LIN {X 0.013,Y -527.446,Z 1176.432,A 0.000,B 0.000,C 90.000,E1 293.695} C_DIS
LIN {X -0.104,Y -527.276,Z 1176.422,A 0.000,B 0.000,C 90.000,E1 291.972} C_DIS
LIN {X -0.041,Y -526.939,Z 1176.411,A 0.000,B 0.000,C 90.000,E1 289.939} C_DIS
LIN {X 0.315,Y -526.514,Z 1176.400,A 0.000,B 0.000,C 90.000,E1 287.873} C_DIS
LIN {X 0.154,Y -526.111,Z 1176.393,A 0.000,B 0.000,C 90.000,E1 286.732} C_DIS
LIN {X -0.007,Y -525.425,Z 1176.385,A 0.000,B 0.000,C 90.000,E1 285.300} C_DIS
LIN {X 0.178,Y -524.796,Z 1176.379,A 0.000,B 0.000,C 90.000,E1 284.120} C_DIS
LIN {X -0.133,Y -523.544,Z 1176.369,A 0.000,B 0.000,C 90.000,E1 282.411} C_DIS
LIN {X -0.073,Y -522.465,Z 1176.359,A 0.000,B 0.000,C 90.000,E1 280.658} C_DIS
LIN {X -0.130,Y -521.579,Z 1176.351,A 0.000,B 0.000,C 90.000,E1 279.208} C_DIS
LIN {X -0.200,Y -520.907,Z 1176.345,A 0.000,B 0.000,C 90.000,E1 278.049} C_DIS
LIN {X 0.164,Y -520.008,Z 1176.337,A 0.000,B 0.000,C 90.000,E1 276.549} C_DIS
LIN {X -0.094,Y -518.805,Z 1176.325,A 0.000,B 0.000,C 90.000,E1 274.531} C_DIS
LIN {X 0.047,Y -517.732,Z 1176.314,A 0.000,B 0.000,C 90.000,E1 272.465} C_DIS
LIN {X 0.205,Y -516.891,Z 1176.304,A 0.000,B 0.000,C 90.000,E1 270.688} C_DIS
LIN {X -0.117,Y -516.202,Z 1176.296,A 0.000,B 0.000,C 90.000,E1 269.255} C_DIS
LIN {X 0.077,Y -515.566,Z 1176.288,A 0.000,B 0.000,C 90.000,E1 267.764} C_DIS
LIN {X -0.182,Y -514.943,Z 1176.281,A 0.000,B 0.000,C 90.000,E1 266.617} C_DIS
LIN {X 0.060,Y -514.072,Z 1176.275,A 0.000,B 0.000,C 90.000,E1 265.412} C_DIS
LIN {X 0.158,Y -512.347,Z 1176.263,A 0.000,B 0.000,C 90.000,E1 263.337} C_DIS
LIN {X -0.115,Y -511.308,Z 1176.257,A 0.000,B 0.000,C 90.000,E1 262.186} C_DIS
LIN {X 0.088,Y -509.594,Z 1176.247,A 0.000,B 0.000,C 90.000,E1 260.387} C_DIS
LIN {X 0.256,Y -507.511,Z 1176.234,A 0.000,B 0.000,C 90.000,E1 257.993} C_DIS
LIN {X 0.024,Y -505.767,Z 1176.222,A 0.000,B 0.000,C 90.000,E1 255.936} C_DIS
LIN {X -0.079,Y -504.700,Z 1176.215,A 0.000,B 0.000,C 90.000,E1 254.755} C_DIS
LIN {X -0.135,Y -503.462,Z 1176.207,A 0.000,B 0.000,C 90.000,E1 253.268} C_DIS
LIN {X 0.005,Y -501.999,Z 1176.197,A 0.000,B 0.000,C 90.000,E1 251.456} C_DIS
LIN {X 0.107,Y -500.375,Z 1176.187,A 0.000,B 0.000,C 90.000,E1 249.645} C_DIS
LIN {X -0.012,Y -498.966,Z 1176.179,A 0.000,B 0.000,C 90.000,E1 248.156} C_DIS
LIN {X -0.149,Y -497.507,Z 1176.170,A 0.000,B 0.000,C 90.000,E1 246.666} C_DIS
LIN {X -0.113,Y -495.810,Z 1176.162,A 0.000,B 0.000,C 90.000,E1 245.153} C_DIS
LIN {X -0.154,Y -494.396,Z 1176.155,A 0.000,B 0.000,C 90.000,E1 243.948} C_DIS
LIN {X 0.036,Y -492.401,Z 1176.147,A 0.000,B 0.000,C 90.000,E1 242.410} C_DIS
LIN {X 0.249,Y -489.559,Z 1176.135,A 0.000,B 0.000,C 90.000,E1 240.255} C_DIS
LIN {X 0.138,Y -487.469,Z 1176.126,A 0.000,B 0.000,C 90.000,E1 238.742} C_DIS
LIN {X 0.051,Y -484.871,Z 1176.116,A 0.000,B 0.000,C 90.000,E1 236.914} C_DIS
LIN {X 0.000,Y -480.986,Z 1176.101,A 0.000,B 0.000,C 90.000,E1 234.149} C_DIS
LIN {X 0.010,Y -478.812,Z 1176.092,A 0.000,B 0.000,C 90.000,E1 232.603} C_DIS
LIN {X -0.040,Y -475.824,Z 1176.080,A 0.000,B 0.000,C 90.000,E1 230.436} C_DIS
LIN {X 0.186,Y -473.842,Z 1176.072,A 0.000,B 0.000,C 90.000,E1 228.852} C_DIS
LIN {X 0.153,Y -472.537,Z 1176.066,A 0.000,B 0.000,C 90.000,E1 227.919} C_DIS
LIN {X -0.220,Y -467.466,Z 1176.047,A 0.000,B 0.000,C 90.000,E1 224.514} C_DIS
LIN {X 0.002,Y -464.713,Z 1176.033,A 0.000,B 0.000,C 90.000,E1 221.962} C_DIS
LIN {X -0.242,Y -462.501,Z 1176.007,A 0.000,B 0.000,C 90.000,E1 217.237} C_DIS
LIN {X 0.183,Y -462.031,Z 1175.991,A 0.000,B 0.000,C 90.000,E1 214.326} C_DIS
LIN {X 0.188,Y -462.258,Z 1175.980,A 0.000,B 0.000,C 90.000,E1 212.418} C_DIS
LIN {X 0.101,Y -463.482,Z 1175.968,A 0.000,B 0.000,C 90.000,E1 210.207} C_DIS
LIN {X 0.219,Y -465.265,Z 1175.956,A 0.000,B 0.000,C 90.000,E1 207.975} C_DIS
LIN {X -0.022,Y -468.504,Z 1175.938,A 0.000,B 0.000,C 90.000,E1 204.847} C_DIS
LIN {X 0.229,Y -475.785,Z 1175.914,A 0.000,B 0.000,C 90.000,E1 200.429} C_DIS
LIN {X 0.047,Y -484.654,Z 1175.893,A 0.000,B 0.000,C 90.000,E1 196.732} C_DIS
LIN {X 0.270,Y -493.798,Z 1175.876,A 0.000,B 0.000,C 90.000,E1 193.647} C_DIS
LIN {X 0.236,Y -500.640,Z 1175.864,A 0.000,B 0.000,C 90.000,E1 191.535} C_DIS
LIN {X -0.107,Y -505.714,Z 1175.856,A 0.000,B 0.000,C 90.000,E1 190.074} C_DIS
LIN {X -0.136,Y -514.040,Z 1175.843,A 0.000,B 0.000,C 90.000,E1 187.701} C_DIS
LIN {X 0.119,Y -519.246,Z 1175.835,A 0.000,B 0.000,C 90.000,E1 186.201} C_DIS
LIN {X -0.147,Y -526.357,Z 1175.823,A 0.000,B 0.000,C 90.000,E1 184.188} C_DIS
LIN {X -0.258,Y -532.477,Z 1175.814,A 0.000,B 0.000,C 90.000,E1 182.465} C_DIS
LIN {X -0.257,Y -539.492,Z 1175.802,A 0.000,B 0.000,C 90.000,E1 180.458} C_DIS
LIN {X -0.180,Y -543.585,Z 1175.796,A 0.000,B 0.000,C 90.000,E1 179.312} C_DIS
LIN {X 0.012,Y -548.578,Z 1175.788,A 0.000,B 0.000,C 90.000,E1 177.879} C_DIS
LIN {X 0.242,Y -552.555,Z 1175.782,A 0.000,B 0.000,C 90.000,E1 176.731} C_DIS
LIN {X 0.160,Y -558.479,Z 1175.773,A 0.000,B 0.000,C 90.000,E1 175.065} C_DIS
LIN {X 0.251,Y -564.346,Z 1175.764,A 0.000,B 0.000,C 90.000,E1 173.394} C_DIS
LIN {X -0.105,Y -570.116,Z 1175.754,A 0.000,B 0.000,C 90.000,E1 171.781} C_DIS
LIN {X 0.183,Y -574.902,Z 1175.747,A 0.000,B 0.000,C 90.000,E1 170.387} C_DIS
LIN {X -0.226,Y -578.690,Z 1175.741,A 0.000,B 0.000,C 90.000,E1 169.342} C_DIS
LIN {X -0.011,Y -584.216,Z 1175.732,A 0.000,B 0.000,C 90.000,E1 167.701} C_DIS
LIN {X 0.069,Y -588.852,Z 1175.724,A 0.000,B 0.000,C 90.000,E1 166.353} C_DIS
LIN {X -0.205,Y -593.226,Z 1175.717,A 0.000,B 0.000,C 90.000,E1 165.046} C_DIS
LIN {X 0.170,Y -597.631,Z 1175.709,A 0.000,B 0.000,C 90.000,E1 163.685} C_DIS
LIN {X -0.073,Y -601.090,Z 1175.704,A 0.000,B 0.000,C 90.000,E1 162.653} C_DIS
LIN {X 0.127,Y -604.447,Z 1175.698,A 0.000,B 0.000,C 90.000,E1 161.583} C_DIS
LIN {X -0.087,Y -608.460,Z 1175.691,A 0.000,B 0.000,C 90.000,E1 160.296} C_DIS
LIN {X 0.351,Y -612.366,Z 1175.683,A 0.000,B 0.000,C 90.000,E1 158.954} C_DIS
LIN {X -0.260,Y -615.395,Z 1175.678,A 0.000,B 0.000,C 90.000,E1 157.975} C_DIS
LIN {X -0.330,Y -620.612,Z 1175.667,A 0.000,B 0.000,C 90.000,E1 156.177} C_DIS
LIN {X 0.220,Y -624.160,Z 1175.660,A 0.000,B 0.000,C 90.000,E1 154.845} C_DIS
LIN {X 0.033,Y -628.945,Z 1175.651,A 0.000,B 0.000,C 90.000,E1 153.076} C_DIS
LIN {X -0.134,Y -631.608,Z 1175.645,A 0.000,B 0.000,C 90.000,E1 152.076} C_DIS
LIN {X 0.040,Y -634.839,Z 1175.638,A 0.000,B 0.000,C 90.000,E1 150.795} C_DIS
LIN {X 0.059,Y -638.466,Z 1175.629,A 0.000,B 0.000,C 90.000,E1 149.282} C_DIS
LIN {X -0.072,Y -641.780,Z 1175.621,A 0.000,B 0.000,C 90.000,E1 147.788} C_DIS
LIN {X -0.056,Y -643.800,Z 1175.615,A 0.000,B 0.000,C 90.000,E1 146.786} C_DIS
LIN {X -0.201,Y -645.736,Z 1175.610,A 0.000,B 0.000,C 90.000,E1 145.801} C_DIS
LIN {X 0.169,Y -648.438,Z 1175.602,A 0.000,B 0.000,C 90.000,E1 144.276} C_DIS
LIN {X 0.007,Y -650.641,Z 1175.595,A 0.000,B 0.000,C 90.000,E1 143.050} C_DIS
LIN {X -0.048,Y -652.350,Z 1175.589,A 0.000,B 0.000,C 90.000,E1 142.065} C_DIS
LIN {X 0.257,Y -654.569,Z 1175.582,A 0.000,B 0.000,C 90.000,E1 140.803} C_DIS
LIN {X 0.097,Y -657.952,Z 1175.573,A 0.000,B 0.000,C 90.000,E1 139.094} C_DIS
LIN {X -0.028,Y -661.068,Z 1175.565,A 0.000,B 0.000,C 90.000,E1 137.634} C_DIS
LIN {X 0.357,Y -664.130,Z 1175.557,A 0.000,B 0.000,C 90.000,E1 136.134} C_DIS
LIN {X 0.346,Y -669.386,Z 1175.543,A 0.000,B 0.000,C 90.000,E1 133.704} C_DIS
LIN {X -0.468,Y -673.988,Z 1175.532,A 0.000,B 0.000,C 90.000,E1 131.838} C_DIS
LIN {X -0.097,Y -679.759,Z 1175.519,A 0.000,B 0.000,C 90.000,E1 129.402} C_DIS
LIN {X -0.135,Y -683.328,Z 1175.511,A 0.000,B 0.000,C 90.000,E1 127.971} C_DIS
LIN {X -0.262,Y -686.330,Z 1175.504,A 0.000,B 0.000,C 90.000,E1 126.790} C_DIS
LIN {X 0.389,Y -689.886,Z 1175.496,A 0.000,B 0.000,C 90.000,E1 125.311} C_DIS
LIN {X -0.098,Y -692.169,Z 1175.491,A 0.000,B 0.000,C 90.000,E1 124.405} C_DIS
LIN {X 0.018,Y -694.299,Z 1175.486,A 0.000,B 0.000,C 90.000,E1 123.452} C_DIS
LIN {X -0.180,Y -696.901,Z 1175.479,A 0.000,B 0.000,C 90.000,E1 122.291} C_DIS
LIN {X 0.000,Y -698.834,Z 1175.474,A 0.000,B 0.000,C 90.000,E1 121.337} C_DIS
LIN {X 0.194,Y -700.659,Z 1175.469,A 0.000,B 0.000,C 90.000,E1 120.384} C_DIS
LIN {X 0.389,Y -701.877,Z 1175.465,A 0.000,B 0.000,C 90.000,E1 119.667} C_DIS
LIN {X -0.074,Y -703.846,Z 1175.459,A 0.000,B 0.000,C 90.000,E1 118.537} C_DIS
LIN {X 0.110,Y -705.271,Z 1175.453,A 0.000,B 0.000,C 90.000,E1 117.590} C_DIS
LIN {X 0.355,Y -706.061,Z 1175.449,A 0.000,B 0.000,C 90.000,E1 116.873} C_DIS
LIN {X -0.051,Y -706.576,Z 1175.444,A 0.000,B 0.000,C 90.000,E1 115.976} C_DIS
LIN {X -0.111,Y -706.732,Z 1175.440,A 0.000,B 0.000,C 90.000,E1 115.283} C_DIS
LIN {X -0.163,Y -706.601,Z 1175.438,A 0.000,B 0.000,C 90.000,E1 114.823} C_DIS
LIN {X -0.165,Y -706.470,Z 1175.437,A 0.000,B 0.000,C 90.000,E1 114.591} C_DIS
LIN {X -0.224,Y -705.621,Z 1175.434,A 0.000,B 0.000,C 90.000,E1 114.131} C_DIS
LIN {X -0.222,Y -705.089,Z 1175.433,A 0.000,B 0.000,C 90.000,E1 113.898} C_DIS
LIN {X -0.434,Y -702.482,Z 1175.429,A 0.000,B 0.000,C 90.000,E1 113.334} C_DIS
LIN {X -0.292,Y -701.641,Z 1175.429,A 0.000,B 0.000,C 90.000,E1 113.206} C_DIS
LIN {X -0.377,Y -697.078,Z 1175.426,A 0.000,B 0.000,C 90.000,E1 112.770} C_DIS
LIN {X -0.200,Y -695.667,Z 1175.426,A 0.000,B 0.000,C 90.000,E1 112.642} C_DIS
LIN {X -0.025,Y -693.336,Z 1175.425,A 0.000,B 0.000,C 90.000,E1 112.514} C_DIS
LIN {X -0.329,Y -686.631,Z 1175.424,A 0.000,B 0.000,C 90.000,E1 112.333} C_DIS
LIN {X -0.052,Y -684.050,Z 1175.424,A 0.000,B 0.000,C 90.000,E1 112.259} C_DIS
LIN {X 0.207,Y -676.815,Z 1175.423,A 0.000,B 0.000,C 90.000,E1 112.206} C_DIS
LIN {X 0.134,Y -605.342,Z 1175.423,A 0.000,B 0.000,C 90.000,E1 112.206} C_DIS
LIN {X -0.130,Y -600.404,Z 1175.422,A 0.000,B 0.000,C 90.000,E1 111.897} C_DIS
LIN {X -0.099,Y -593.606,Z 1175.419,A 0.000,B 0.000,C 90.000,E1 111.354} C_DIS
LIN {X 0.310,Y -585.303,Z 1175.415,A 0.000,B 0.000,C 90.000,E1 110.610} C_DIS
LIN {X 0.237,Y -575.542,Z 1175.410,A 0.000,B 0.000,C 90.000,E1 109.812} C_DIS
LIN {X 0.038,Y -567.954,Z 1175.407,A 0.000,B 0.000,C 90.000,E1 109.268} C_DIS
LIN {X 0.086,Y -555.843,Z 1175.402,A 0.000,B 0.000,C 90.000,E1 108.417} C_DIS
LIN {X -0.159,Y -552.031,Z 1175.401,A 0.000,B 0.000,C 90.000,E1 108.109} C_DIS
LIN {X -0.164,Y -550.794,Z 1175.399,A 0.000,B 0.000,C 90.000,E1 107.873} C_DIS
LIN {X 0.140,Y -550.193,Z 1175.397,A 0.000,B 0.000,C 90.000,E1 107.457} C_DIS
LIN {X -0.210,Y -550.647,Z 1175.392,A 0.000,B 0.000,C 90.000,E1 106.496} C_DIS
LIN {X 0.083,Y -551.869,Z 1175.384,A 0.000,B 0.000,C 90.000,E1 105.064} C_DIS
LIN {X 0.255,Y -553.162,Z 1175.376,A 0.000,B 0.000,C 90.000,E1 103.647} C_DIS
LIN {X 0.041,Y -554.958,Z 1175.365,A 0.000,B 0.000,C 90.000,E1 101.715} C_DIS
LIN {X -0.134,Y -557.005,Z 1175.354,A 0.000,B 0.000,C 90.000,E1 99.782} C_DIS
LIN {X -0.044,Y -558.660,Z 1175.345,A 0.000,B 0.000,C 90.000,E1 98.106} C_DIS
LIN {X -0.124,Y -559.628,Z 1175.339,A 0.000,B 0.000,C 90.000,E1 97.004} C_DIS
LIN {X -0.181,Y -560.682,Z 1175.331,A 0.000,B 0.000,C 90.000,E1 95.625} C_DIS
LIN {X 0.012,Y -561.969,Z 1175.320,A 0.000,B 0.000,C 90.000,E1 93.669} C_DIS
LIN {X -0.270,Y -563.607,Z 1175.308,A 0.000,B 0.000,C 90.000,E1 91.489} C_DIS
LIN {X 0.263,Y -564.658,Z 1175.301,A 0.000,B 0.000,C 90.000,E1 90.057} C_DIS
LIN {X 0.253,Y -565.605,Z 1175.293,A 0.000,B 0.000,C 90.000,E1 88.682} C_DIS
LIN {X -0.183,Y -566.714,Z 1175.284,A 0.000,B 0.000,C 90.000,E1 87.078} C_DIS
LIN {X 0.157,Y -567.924,Z 1175.273,A 0.000,B 0.000,C 90.000,E1 85.122} C_DIS
LIN {X 0.255,Y -568.879,Z 1175.265,A 0.000,B 0.000,C 90.000,E1 83.742} C_DIS
LIN {X -0.033,Y -570.009,Z 1175.256,A 0.000,B 0.000,C 90.000,E1 82.129} C_DIS
LIN {X 0.235,Y -570.783,Z 1175.249,A 0.000,B 0.000,C 90.000,E1 80.735} C_DIS
LIN {X -0.218,Y -571.811,Z 1175.238,A 0.000,B 0.000,C 90.000,E1 78.870} C_DIS
LIN {X -0.166,Y -572.642,Z 1175.229,A 0.000,B 0.000,C 90.000,E1 77.229} C_DIS
LIN {X 0.035,Y -573.494,Z 1175.220,A 0.000,B 0.000,C 90.000,E1 75.574} C_DIS
LIN {X -0.295,Y -574.029,Z 1175.214,A 0.000,B 0.000,C 90.000,E1 74.519} C_DIS
LIN {X 0.070,Y -575.221,Z 1175.202,A 0.000,B 0.000,C 90.000,E1 72.308} C_DIS
LIN {X -0.087,Y -576.420,Z 1175.191,A 0.000,B 0.000,C 90.000,E1 70.423} C_DIS
LIN {X -0.226,Y -577.390,Z 1175.184,A 0.000,B 0.000,C 90.000,E1 69.082} C_DIS
LIN {X 0.114,Y -579.685,Z 1175.170,A 0.000,B 0.000,C 90.000,E1 66.613} C_DIS
LIN {X 0.078,Y -580.709,Z 1175.164,A 0.000,B 0.000,C 90.000,E1 65.537} C_DIS
LIN {X 0.321,Y -582.243,Z 1175.155,A 0.000,B 0.000,C 90.000,E1 63.896} C_DIS
LIN {X 0.058,Y -583.760,Z 1175.146,A 0.000,B 0.000,C 90.000,E1 62.308} C_DIS
LIN {X -0.144,Y -585.299,Z 1175.137,A 0.000,B 0.000,C 90.000,E1 60.717} C_DIS
LIN {X 0.327,Y -586.452,Z 1175.130,A 0.000,B 0.000,C 90.000,E1 59.331} C_DIS
LIN {X 0.311,Y -587.524,Z 1175.122,A 0.000,B 0.000,C 90.000,E1 57.995} C_DIS
LIN {X -0.127,Y -588.870,Z 1175.112,A 0.000,B 0.000,C 90.000,E1 56.167} C_DIS
LIN {X -0.085,Y -589.941,Z 1175.103,A 0.000,B 0.000,C 90.000,E1 54.562} C_DIS
LIN {X -0.146,Y -590.960,Z 1175.094,A 0.000,B 0.000,C 90.000,E1 52.970} C_DIS
LIN {X 0.035,Y -592.084,Z 1175.084,A 0.000,B 0.000,C 90.000,E1 51.090} C_DIS
LIN {X -0.031,Y -592.648,Z 1175.078,A 0.000,B 0.000,C 90.000,E1 50.033} C_DIS
LIN {X 0.126,Y -593.129,Z 1175.071,A 0.000,B 0.000,C 90.000,E1 48.690} C_DIS
LIN {X 0.069,Y -593.403,Z 1175.065,A 0.000,B 0.000,C 90.000,E1 47.634} C_DIS
LIN {X 0.181,Y -593.608,Z 1175.057,A 0.000,B 0.000,C 90.000,E1 46.296} C_DIS
LIN {X -0.130,Y -593.404,Z 1175.050,A 0.000,B 0.000,C 90.000,E1 45.000} C_DIS
LIN {X -0.213,Y -593.146,Z 1175.044,A 0.000,B 0.000,C 90.000,E1 43.947} C_DIS
LIN {X 0.128,Y -592.599,Z 1175.038,A 0.000,B 0.000,C 90.000,E1 42.852} C_DIS
LIN {X 0.220,Y -591.768,Z 1175.031,A 0.000,B 0.000,C 90.000,E1 41.515} C_DIS
LIN {X -0.061,Y -591.167,Z 1175.026,A 0.000,B 0.000,C 90.000,E1 40.744} C_DIS
LIN {X 0.052,Y -589.816,Z 1175.019,A 0.000,B 0.000,C 90.000,E1 39.402} C_DIS
LIN {X -0.168,Y -588.919,Z 1175.015,A 0.000,B 0.000,C 90.000,E1 38.624} C_DIS
LIN {X -0.097,Y -587.117,Z 1175.007,A 0.000,B 0.000,C 90.000,E1 37.282} C_DIS
LIN {X -0.146,Y -585.336,Z 1175.001,A 0.000,B 0.000,C 90.000,E1 36.217} C_DIS
LIN {X 0.258,Y -583.221,Z 1174.995,A 0.000,B 0.000,C 90.000,E1 35.105} C_DIS
LIN {X -0.194,Y -581.990,Z 1174.992,A 0.000,B 0.000,C 90.000,E1 34.612} C_DIS
LIN {X -0.004,Y -579.896,Z 1174.988,A 0.000,B 0.000,C 90.000,E1 33.785} C_DIS
LIN {X 0.164,Y -577.455,Z 1174.983,A 0.000,B 0.000,C 90.000,E1 32.959} C_DIS
LIN {X 0.302,Y -574.678,Z 1174.979,A 0.000,B 0.000,C 90.000,E1 32.133} C_DIS
LIN {X 0.105,Y -571.556,Z 1174.974,A 0.000,B 0.000,C 90.000,E1 31.337} C_DIS
LIN {X -0.031,Y -568.604,Z 1174.970,A 0.000,B 0.000,C 90.000,E1 30.669} C_DIS
LIN {X -0.194,Y -565.352,Z 1174.967,A 0.000,B 0.000,C 90.000,E1 30.001} C_DIS
LIN {X 0.198,Y -562.567,Z 1174.964,A 0.000,B 0.000,C 90.000,E1 29.411} C_DIS
LIN {X -0.230,Y -557.191,Z 1174.958,A 0.000,B 0.000,C 90.000,E1 28.487} C_DIS
LIN {X -0.122,Y -552.159,Z 1174.953,A 0.000,B 0.000,C 90.000,E1 27.641} C_DIS
LIN {X 0.030,Y -549.475,Z 1174.951,A 0.000,B 0.000,C 90.000,E1 27.206} C_DIS
LIN {X 0.174,Y -544.626,Z 1174.947,A 0.000,B 0.000,C 90.000,E1 26.488} C_DIS
LIN {X 0.032,Y -539.444,Z 1174.943,A 0.000,B 0.000,C 90.000,E1 25.796} C_DIS
LIN {X 0.202,Y -533.965,Z 1174.939,A 0.000,B 0.000,C 90.000,E1 25.079} C_DIS
LIN {X 0.147,Y -525.389,Z 1174.934,A 0.000,B 0.000,C 90.000,E1 24.079} C_DIS
LIN {X 0.021,Y -520.243,Z 1174.931,A 0.000,B 0.000,C 90.000,E1 23.515} C_DIS
LIN {X 0.038,Y -513.748,Z 1174.927,A 0.000,B 0.000,C 90.000,E1 22.823} C_DIS
LIN {X 0.174,Y -505.611,Z 1174.922,A 0.000,B 0.000,C 90.000,E1 21.972} C_DIS
LIN {X -0.183,Y -500.013,Z 1174.919,A 0.000,B 0.000,C 90.000,E1 21.461} C_DIS
LIN {X 0.117,Y -488.798,Z 1174.913,A 0.000,B 0.000,C 90.000,E1 20.375} C_DIS
LIN {X 0.092,Y -477.040,Z 1174.907,A 0.000,B 0.000,C 90.000,E1 19.322} C_DIS
LIN {X 0.050,Y -469.683,Z 1174.904,A 0.000,B 0.000,C 90.000,E1 18.671} C_DIS
LIN {X -0.113,Y -462.529,Z 1174.900,A 0.000,B 0.000,C 90.000,E1 18.055} C_DIS
LIN {X -0.066,Y -437.599,Z 1174.887,A 0.000,B 0.000,C 90.000,E1 15.717} C_DIS
LIN {X 0.172,Y -424.699,Z 1174.880,A 0.000,B 0.000,C 90.000,E1 14.356} C_DIS
LIN {X 0.113,Y -412.177,Z 1174.872,A 0.000,B 0.000,C 90.000,E1 12.939} C_DIS
LIN {X 0.147,Y -401.660,Z 1174.865,A 0.000,B 0.000,C 90.000,E1 11.591} C_DIS
LIN {X 0.130,Y -396.838,Z 1174.861,A 0.000,B 0.000,C 90.000,E1 10.894} C_DIS
LIN {X 0.127,Y -394.011,Z 1174.858,A 0.000,B 0.000,C 90.000,E1 10.366} C_DIS
LIN {X 0.024,Y -392.896,Z 1174.855,A 0.000,B 0.000,C 90.000,E1 9.962} C_DIS
LIN {X -0.015,Y -392.883,Z 1174.855,A 0.000,B 0.000,C 90.000,E1 9.962} C_DIS
LIN {X -0.002,Y -393.309,Z 1174.853,A 0.000,B 0.000,C 90.000,E1 9.500} C_DIS
LIN {X -0.135,Y -394.602,Z 1174.850,A 0.000,B 0.000,C 90.000,E1 8.973} C_DIS
LIN {X -0.145,Y -396.919,Z 1174.846,A 0.000,B 0.000,C 90.000,E1 8.276} C_DIS
LIN {X 0.216,Y -398.327,Z 1174.844,A 0.000,B 0.000,C 90.000,E1 7.871} C_DIS
LIN {X -0.191,Y -402.030,Z 1174.839,A 0.000,B 0.000,C 90.000,E1 7.125} C_DIS
LIN {X 0.193,Y -406.606,Z 1174.836,A 0.000,B 0.000,C 90.000,E1 6.429} C_DIS
LIN {X -0.021,Y -407.352,Z 1174.835,A 0.000,B 0.000,C 90.000,E1 6.372} C_DIS
LIN {X 0.169,Y -411.554,Z 1174.833,A 0.000,B 0.000,C 90.000,E1 5.967} C_DIS
LIN {X -0.196,Y -429.455,Z 1174.826,A 0.000,B 0.000,C 90.000,E1 4.645} C_DIS
LIN {X -0.050,Y -450.379,Z 1174.817,A 0.000,B 0.000,C 90.000,E1 3.094} C_DIS
LIN {X 0.092,Y -464.698,Z 1174.812,A 0.000,B 0.000,C 90.000,E1 2.064} C_DIS
LIN {X 0.128,Y -472.596,Z 1174.808,A 0.000,B 0.000,C 90.000,E1 1.489} C_DIS
LIN {X 0.165,Y -480.262,Z 1174.805,A 0.000,B 0.000,C 90.000,E1 0.917} C_DIS
LIN {X 0.097,Y -484.863,Z 1174.803,A 0.000,B 0.000,C 90.000,E1 0.573} C_DIS
LIN {X -0.110,Y -490.882,Z 1174.801,A 0.000,B 0.000,C 90.000,E1 0.115} C_DIS
LIN {X 0.118,Y -497.274,Z 1174.798,A 0.000,B 0.000,C 90.000,E1 359.542} C_DIS
LIN {X -0.077,Y -504.181,Z 1174.794,A 0.000,B 0.000,C 90.000,E1 358.912} C_DIS
LIN {X -0.140,Y -510.853,Z 1174.790,A 0.000,B 0.000,C 90.000,E1 358.224} C_DIS
LIN {X 0.111,Y -517.176,Z 1174.786,A 0.000,B 0.000,C 90.000,E1 357.478} C_DIS
LIN {X 0.259,Y -523.171,Z 1174.782,A 0.000,B 0.000,C 90.000,E1 356.731} C_DIS
LIN {X -0.006,Y -528.449,Z 1174.778,A 0.000,B 0.000,C 90.000,E1 356.045} C_DIS
LIN {X -0.028,Y -532.451,Z 1174.775,A 0.000,B 0.000,C 90.000,E1 355.469} C_DIS
LIN {X 0.243,Y -536.965,Z 1174.771,A 0.000,B 0.000,C 90.000,E1 354.723} C_DIS
LIN {X 0.020,Y -540.996,Z 1174.767,A 0.000,B 0.000,C 90.000,E1 354.033} C_DIS
LIN {X 0.091,Y -543.955,Z 1174.764,A 0.000,B 0.000,C 90.000,E1 353.457} C_DIS
LIN {X -0.012,Y -547.296,Z 1174.760,A 0.000,B 0.000,C 90.000,E1 352.761} C_DIS
LIN {X 0.105,Y -549.791,Z 1174.757,A 0.000,B 0.000,C 90.000,E1 352.186} C_DIS
LIN {X -0.232,Y -552.111,Z 1174.754,A 0.000,B 0.000,C 90.000,E1 351.659} C_DIS
LIN {X 0.033,Y -555.204,Z 1174.749,A 0.000,B 0.000,C 90.000,E1 350.792} C_DIS
LIN {X 0.195,Y -557.124,Z 1174.746,A 0.000,B 0.000,C 90.000,E1 350.218} C_DIS
LIN {X 0.056,Y -559.719,Z 1174.741,A 0.000,B 0.000,C 90.000,E1 349.398} C_DIS
LIN {X -0.051,Y -562.098,Z 1174.737,A 0.000,B 0.000,C 90.000,E1 348.578} C_DIS
LIN {X -0.130,Y -564.331,Z 1174.732,A 0.000,B 0.000,C 90.000,E1 347.757} C_DIS
LIN {X -0.018,Y -567.166,Z 1174.726,A 0.000,B 0.000,C 90.000,E1 346.645} C_DIS
LIN {X 0.075,Y -571.006,Z 1174.717,A 0.000,B 0.000,C 90.000,E1 344.991} C_DIS
LIN {X -0.139,Y -573.412,Z 1174.711,A 0.000,B 0.000,C 90.000,E1 343.921} C_DIS
LIN {X -0.323,Y -576.785,Z 1174.702,A 0.000,B 0.000,C 90.000,E1 342.308} C_DIS
LIN {X 0.089,Y -579.327,Z 1174.694,A 0.000,B 0.000,C 90.000,E1 340.913} C_DIS
LIN {X 0.004,Y -581.559,Z 1174.687,A 0.000,B 0.000,C 90.000,E1 339.571} C_DIS
LIN {X -0.097,Y -582.756,Z 1174.682,A 0.000,B 0.000,C 90.000,E1 338.773} C_DIS
LIN {X 0.087,Y -584.321,Z 1174.675,A 0.000,B 0.000,C 90.000,E1 337.411} C_DIS
LIN {X 0.010,Y -584.904,Z 1174.670,A 0.000,B 0.000,C 90.000,E1 336.613} C_DIS
LIN {X 0.046,Y -585.271,Z 1174.664,A 0.000,B 0.000,C 90.000,E1 335.537} C_DIS
LIN {X 0.212,Y -585.052,Z 1174.660,A 0.000,B 0.000,C 90.000,E1 334.717} C_DIS
LIN {X -0.152,Y -584.598,Z 1174.655,A 0.000,B 0.000,C 90.000,E1 333.948} C_DIS
LIN {X 0.128,Y -584.149,Z 1174.652,A 0.000,B 0.000,C 90.000,E1 333.384} C_DIS
LIN {X -0.247,Y -583.036,Z 1174.648,A 0.000,B 0.000,C 90.000,E1 332.615} C_DIS
LIN {X 0.022,Y -581.106,Z 1174.642,A 0.000,B 0.000,C 90.000,E1 331.513} C_DIS
LIN {X -0.107,Y -579.179,Z 1174.637,A 0.000,B 0.000,C 90.000,E1 330.717} C_DIS
LIN {X -0.105,Y -577.738,Z 1174.634,A 0.000,B 0.000,C 90.000,E1 330.177} C_DIS
LIN {X 0.097,Y -576.016,Z 1174.631,A 0.000,B 0.000,C 90.000,E1 329.616} C_DIS
LIN {X -0.005,Y -573.435,Z 1174.628,A 0.000,B 0.000,C 90.000,E1 328.948} C_DIS
LIN {X 0.080,Y -569.210,Z 1174.623,A 0.000,B 0.000,C 90.000,E1 328.122} C_DIS
LIN {X 0.014,Y -566.137,Z 1174.620,A 0.000,B 0.000,C 90.000,E1 327.582} C_DIS
LIN {X -0.080,Y -559.740,Z 1174.615,A 0.000,B 0.000,C 90.000,E1 326.628} C_DIS
LIN {X -0.101,Y -556.739,Z 1174.612,A 0.000,B 0.000,C 90.000,E1 326.215} C_DIS
LIN {X -0.255,Y -552.404,Z 1174.609,A 0.000,B 0.000,C 90.000,E1 325.674} C_DIS
LIN {X -0.077,Y -545.498,Z 1174.604,A 0.000,B 0.000,C 90.000,E1 324.815} C_DIS
LIN {X -0.139,Y -539.228,Z 1174.601,A 0.000,B 0.000,C 90.000,E1 324.116} C_DIS
LIN {X -0.036,Y -526.801,Z 1174.593,A 0.000,B 0.000,C 90.000,E1 322.718} C_DIS
LIN {X -0.061,Y -524.415,Z 1174.591,A 0.000,B 0.000,C 90.000,E1 322.431} C_DIS
LIN {X 0.045,Y -521.309,Z 1174.589,A 0.000,B 0.000,C 90.000,E1 321.984} C_DIS
LIN {X 0.031,Y -518.478,Z 1174.586,A 0.000,B 0.000,C 90.000,E1 321.492} C_DIS
LIN {X 0.057,Y -516.504,Z 1174.583,A 0.000,B 0.000,C 90.000,E1 320.884} C_DIS
LIN {X 0.251,Y -515.793,Z 1174.579,A 0.000,B 0.000,C 90.000,E1 320.275} C_DIS
LIN {X 0.109,Y -515.594,Z 1174.576,A 0.000,B 0.000,C 90.000,E1 319.703} C_DIS
LIN {X 0.213,Y -516.613,Z 1174.565,A 0.000,B 0.000,C 90.000,E1 317.634} C_DIS
LIN {X -0.040,Y -517.789,Z 1174.553,A 0.000,B 0.000,C 90.000,E1 315.607} C_DIS
LIN {X 0.260,Y -518.623,Z 1174.545,A 0.000,B 0.000,C 90.000,E1 314.109} C_DIS
LIN {X 0.135,Y -519.616,Z 1174.536,A 0.000,B 0.000,C 90.000,E1 312.366} C_DIS
LIN {X 0.065,Y -520.722,Z 1174.526,A 0.000,B 0.000,C 90.000,E1 310.620} C_DIS
LIN {X -0.214,Y -521.451,Z 1174.519,A 0.000,B 0.000,C 90.000,E1 309.483} C_DIS
LIN {X -0.222,Y -522.748,Z 1174.508,A 0.000,B 0.000,C 90.000,E1 307.443} C_DIS
LIN {X -0.011,Y -523.514,Z 1174.500,A 0.000,B 0.000,C 90.000,E1 305.964} C_DIS
LIN {X 0.098,Y -524.829,Z 1174.487,A 0.000,B 0.000,C 90.000,E1 303.627} C_DIS
LIN {X -0.238,Y -525.703,Z 1174.479,A 0.000,B 0.000,C 90.000,E1 302.212} C_DIS
LIN {X -0.148,Y -526.586,Z 1174.469,A 0.000,B 0.000,C 90.000,E1 300.463} C_DIS
LIN {X -0.052,Y -526.883,Z 1174.466,A 0.000,B 0.000,C 90.000,E1 299.873} C_DIS
LIN {X 0.253,Y -527.409,Z 1174.456,A 0.000,B 0.000,C 90.000,E1 298.103} C_DIS
LIN {X -0.154,Y -527.708,Z 1174.447,A 0.000,B 0.000,C 90.000,E1 296.411} C_DIS
LIN {X 0.282,Y -527.875,Z 1174.440,A 0.000,B 0.000,C 90.000,E1 295.207} C_DIS
LIN {X 0.200,Y -527.883,Z 1174.432,A 0.000,B 0.000,C 90.000,E1 293.770} C_DIS
LIN {X -0.190,Y -527.721,Z 1174.423,A 0.000,B 0.000,C 90.000,E1 292.078} C_DIS
LIN {X 0.192,Y -527.431,Z 1174.413,A 0.000,B 0.000,C 90.000,E1 290.301} C_DIS
LIN {X 0.063,Y -526.927,Z 1174.400,A 0.000,B 0.000,C 90.000,E1 288.000} C_DIS
LIN {X -0.087,Y -526.526,Z 1174.394,A 0.000,B 0.000,C 90.000,E1 286.858} C_DIS
LIN {X 0.257,Y -526.045,Z 1174.387,A 0.000,B 0.000,C 90.000,E1 285.662} C_DIS
LIN {X -0.038,Y -525.275,Z 1174.379,A 0.000,B 0.000,C 90.000,E1 284.245} C_DIS
LIN {X 0.181,Y -524.054,Z 1174.370,A 0.000,B 0.000,C 90.000,E1 282.479} C_DIS
LIN {X -0.261,Y -523.182,Z 1174.361,A 0.000,B 0.000,C 90.000,E1 281.074} C_DIS
LIN {X -0.203,Y -522.038,Z 1174.352,A 0.000,B 0.000,C 90.000,E1 279.321} C_DIS
LIN {X 0.245,Y -521.372,Z 1174.345,A 0.000,B 0.000,C 90.000,E1 278.106} C_DIS
LIN {X 0.098,Y -520.485,Z 1174.337,A 0.000,B 0.000,C 90.000,E1 276.663} C_DIS
LIN {X -0.212,Y -519.099,Z 1174.324,A 0.000,B 0.000,C 90.000,E1 274.359} C_DIS
LIN {X 0.001,Y -518.252,Z 1174.314,A 0.000,B 0.000,C 90.000,E1 272.579} C_DIS
LIN {X 0.107,Y -517.224,Z 1174.303,A 0.000,B 0.000,C 90.000,E1 270.516} C_DIS
LIN {X 0.243,Y -516.461,Z 1174.293,A 0.000,B 0.000,C 90.000,E1 268.740} C_DIS
LIN {X -0.076,Y -515.815,Z 1174.285,A 0.000,B 0.000,C 90.000,E1 267.306} C_DIS
LIN {X 0.178,Y -515.105,Z 1174.279,A 0.000,B 0.000,C 90.000,E1 266.102} C_DIS
LIN {X -0.056,Y -514.156,Z 1174.272,A 0.000,B 0.000,C 90.000,E1 264.951} C_DIS
LIN {X 0.049,Y -512.436,Z 1174.260,A 0.000,B 0.000,C 90.000,E1 262.875} C_DIS
LIN {X -0.225,Y -511.314,Z 1174.254,A 0.000,B 0.000,C 90.000,E1 261.724} C_DIS
LIN {X -0.065,Y -509.345,Z 1174.242,A 0.000,B 0.000,C 90.000,E1 259.634} C_DIS
LIN {X 0.197,Y -507.337,Z 1174.229,A 0.000,B 0.000,C 90.000,E1 257.229} C_DIS
LIN {X -0.043,Y -505.588,Z 1174.218,A 0.000,B 0.000,C 90.000,E1 255.172} C_DIS
LIN {X -0.009,Y -504.017,Z 1174.208,A 0.000,B 0.000,C 90.000,E1 253.378} C_DIS
LIN {X 0.068,Y -502.282,Z 1174.196,A 0.000,B 0.000,C 90.000,E1 251.275} C_DIS
LIN {X -0.293,Y -500.596,Z 1174.186,A 0.000,B 0.000,C 90.000,E1 249.518} C_DIS
LIN {X -0.010,Y -499.538,Z 1174.179,A 0.000,B 0.000,C 90.000,E1 248.284} C_DIS
LIN {X -0.077,Y -497.728,Z 1174.169,A 0.000,B 0.000,C 90.000,E1 246.485} C_DIS
LIN {X 0.009,Y -495.623,Z 1174.159,A 0.000,B 0.000,C 90.000,E1 244.665} C_DIS
LIN {X -0.083,Y -494.526,Z 1174.154,A 0.000,B 0.000,C 90.000,E1 243.768} C_DIS
LIN {X 0.104,Y -492.490,Z 1174.146,A 0.000,B 0.000,C 90.000,E1 242.231} C_DIS
LIN {X 0.058,Y -490.027,Z 1174.136,A 0.000,B 0.000,C 90.000,E1 240.411} C_DIS
LIN {X 0.200,Y -487.941,Z 1174.127,A 0.000,B 0.000,C 90.000,E1 238.869} C_DIS
LIN {X 0.126,Y -485.329,Z 1174.117,A 0.000,B 0.000,C 90.000,E1 237.041} C_DIS
LIN {X 0.098,Y -481.399,Z 1174.102,A 0.000,B 0.000,C 90.000,E1 234.276} C_DIS
LIN {X 0.019,Y -479.666,Z 1174.095,A 0.000,B 0.000,C 90.000,E1 233.050} C_DIS
LIN {X -0.280,Y -477.463,Z 1174.086,A 0.000,B 0.000,C 90.000,E1 231.537} C_DIS
LIN {X 0.230,Y -474.561,Z 1174.074,A 0.000,B 0.000,C 90.000,E1 229.299} C_DIS
LIN {X -0.015,Y -472.915,Z 1174.067,A 0.000,B 0.000,C 90.000,E1 228.081} C_DIS
LIN {X -0.202,Y -470.361,Z 1174.058,A 0.000,B 0.000,C 90.000,E1 226.539} C_DIS
LIN {X -0.018,Y -465.761,Z 1174.039,A 0.000,B 0.000,C 90.000,E1 223.056} C_DIS
LIN {X 0.221,Y -462.844,Z 1174.016,A 0.000,B 0.000,C 90.000,E1 218.910} C_DIS
LIN {X 0.023,Y -462.311,Z 1174.006,A 0.000,B 0.000,C 90.000,E1 217.030} C_DIS
LIN {X -0.201,Y -461.792,Z 1173.990,A 0.000,B 0.000,C 90.000,E1 214.199} C_DIS
LIN {X 0.050,Y -461.970,Z 1173.979,A 0.000,B 0.000,C 90.000,E1 212.260} C_DIS
LIN {X -0.016,Y -463.660,Z 1173.963,A 0.000,B 0.000,C 90.000,E1 209.411} C_DIS
LIN {X -0.047,Y -466.061,Z 1173.948,A 0.000,B 0.000,C 90.000,E1 206.565} C_DIS
LIN {X 0.077,Y -469.105,Z 1173.934,A 0.000,B 0.000,C 90.000,E1 204.027} C_DIS
LIN {X 0.209,Y -476.318,Z 1173.911,A 0.000,B 0.000,C 90.000,E1 199.939} C_DIS
LIN {X 0.050,Y -484.705,Z 1173.892,A 0.000,B 0.000,C 90.000,E1 196.551} C_DIS
LIN {X 0.157,Y -493.971,Z 1173.875,A 0.000,B 0.000,C 90.000,E1 193.480} C_DIS
LIN {X 0.139,Y -500.904,Z 1173.863,A 0.000,B 0.000,C 90.000,E1 191.366} C_DIS
LIN {X -0.251,Y -507.007,Z 1173.853,A 0.000,B 0.000,C 90.000,E1 189.613} C_DIS
LIN {X -0.206,Y -514.402,Z 1173.842,A 0.000,B 0.000,C 90.000,E1 187.530} C_DIS
LIN {X 0.136,Y -518.595,Z 1173.835,A 0.000,B 0.000,C 90.000,E1 186.315} C_DIS
LIN {X -0.149,Y -525.752,Z 1173.824,A 0.000,B 0.000,C 90.000,E1 184.302} C_DIS
LIN {X 0.257,Y -531.928,Z 1173.814,A 0.000,B 0.000,C 90.000,E1 182.522} C_DIS
LIN {X 0.242,Y -537.954,Z 1173.805,A 0.000,B 0.000,C 90.000,E1 180.802} C_DIS
LIN {X -0.193,Y -544.114,Z 1173.795,A 0.000,B 0.000,C 90.000,E1 179.141} C_DIS
LIN {X 0.009,Y -549.165,Z 1173.787,A 0.000,B 0.000,C 90.000,E1 177.707} C_DIS
LIN {X -0.247,Y -554.138,Z 1173.780,A 0.000,B 0.000,C 90.000,E1 176.331} C_DIS
LIN {X 0.247,Y -560.110,Z 1173.770,A 0.000,B 0.000,C 90.000,E1 174.609} C_DIS
LIN {X 0.274,Y -565.036,Z 1173.763,A 0.000,B 0.000,C 90.000,E1 173.223} C_DIS
LIN {X -0.171,Y -569.911,Z 1173.755,A 0.000,B 0.000,C 90.000,E1 171.894} C_DIS
LIN {X -0.142,Y -576.674,Z 1173.744,A 0.000,B 0.000,C 90.000,E1 169.982} C_DIS
LIN {X 0.147,Y -580.428,Z 1173.738,A 0.000,B 0.000,C 90.000,E1 168.870} C_DIS
LIN {X 0.168,Y -585.112,Z 1173.731,A 0.000,B 0.000,C 90.000,E1 167.521} C_DIS
LIN {X 0.269,Y -589.750,Z 1173.723,A 0.000,B 0.000,C 90.000,E1 166.172} C_DIS
LIN {X -0.016,Y -595.924,Z 1173.713,A 0.000,B 0.000,C 90.000,E1 164.338} C_DIS
LIN {X 0.288,Y -601.164,Z 1173.704,A 0.000,B 0.000,C 90.000,E1 162.725} C_DIS
LIN {X 0.099,Y -604.532,Z 1173.698,A 0.000,B 0.000,C 90.000,E1 161.692} C_DIS
LIN {X -0.237,Y -607.774,Z 1173.693,A 0.000,B 0.000,C 90.000,E1 160.678} C_DIS
LIN {X 0.125,Y -612.421,Z 1173.684,A 0.000,B 0.000,C 90.000,E1 159.082} C_DIS
LIN {X 0.082,Y -615.452,Z 1173.678,A 0.000,B 0.000,C 90.000,E1 158.050} C_DIS
LIN {X 0.257,Y -620.633,Z 1173.668,A 0.000,B 0.000,C 90.000,E1 156.230} C_DIS
LIN {X -0.015,Y -624.167,Z 1173.661,A 0.000,B 0.000,C 90.000,E1 154.973} C_DIS
LIN {X 0.060,Y -628.214,Z 1173.652,A 0.000,B 0.000,C 90.000,E1 153.435} C_DIS
LIN {X 0.186,Y -631.586,Z 1173.645,A 0.000,B 0.000,C 90.000,E1 152.153} C_DIS
LIN {X -0.198,Y -634.754,Z 1173.638,A 0.000,B 0.000,C 90.000,E1 150.923} C_DIS
LIN {X -0.226,Y -637.778,Z 1173.631,A 0.000,B 0.000,C 90.000,E1 149.665} C_DIS
LIN {X 0.181,Y -641.130,Z 1173.623,A 0.000,B 0.000,C 90.000,E1 148.122} C_DIS
LIN {X 0.192,Y -643.248,Z 1173.617,A 0.000,B 0.000,C 90.000,E1 147.120} C_DIS
LIN {X 0.095,Y -645.614,Z 1173.611,A 0.000,B 0.000,C 90.000,E1 145.881} C_DIS
LIN {X -0.016,Y -648.721,Z 1173.601,A 0.000,B 0.000,C 90.000,E1 144.149} C_DIS
LIN {X 0.261,Y -651.365,Z 1173.593,A 0.000,B 0.000,C 90.000,E1 142.637} C_DIS
LIN {X 0.027,Y -654.392,Z 1173.583,A 0.000,B 0.000,C 90.000,E1 140.928} C_DIS
LIN {X 0.334,Y -658.226,Z 1173.572,A 0.000,B 0.000,C 90.000,E1 138.933} C_DIS
LIN {X 0.240,Y -660.822,Z 1173.565,A 0.000,B 0.000,C 90.000,E1 137.715} C_DIS
LIN {X -0.317,Y -663.896,Z 1173.557,A 0.000,B 0.000,C 90.000,E1 136.296} C_DIS
LIN {X -0.342,Y -669.105,Z 1173.544,A 0.000,B 0.000,C 90.000,E1 133.866} C_DIS
LIN {X -0.214,Y -673.711,Z 1173.533,A 0.000,B 0.000,C 90.000,E1 131.919} C_DIS
LIN {X -0.252,Y -680.086,Z 1173.518,A 0.000,B 0.000,C 90.000,E1 129.277} C_DIS
LIN {X -0.212,Y -684.861,Z 1173.508,A 0.000,B 0.000,C 90.000,E1 127.363} C_DIS
LIN {X -0.149,Y -688.390,Z 1173.500,A 0.000,B 0.000,C 90.000,E1 125.931} C_DIS
LIN {X -0.062,Y -691.338,Z 1173.493,A 0.000,B 0.000,C 90.000,E1 124.739} C_DIS
LIN {X -0.316,Y -694.047,Z 1173.486,A 0.000,B 0.000,C 90.000,E1 123.579} C_DIS
LIN {X 0.440,Y -696.665,Z 1173.480,A 0.000,B 0.000,C 90.000,E1 122.339} C_DIS
LIN {X -0.005,Y -698.144,Z 1173.476,A 0.000,B 0.000,C 90.000,E1 121.671} C_DIS
LIN {X -0.159,Y -700.424,Z 1173.469,A 0.000,B 0.000,C 90.000,E1 120.512} C_DIS
LIN {X 0.032,Y -701.699,Z 1173.466,A 0.000,B 0.000,C 90.000,E1 119.795} C_DIS
LIN {X 0.182,Y -703.692,Z 1173.459,A 0.000,B 0.000,C 90.000,E1 118.615} C_DIS
LIN {X 0.033,Y -705.468,Z 1173.453,A 0.000,B 0.000,C 90.000,E1 117.462} C_DIS
LIN {X 0.279,Y -706.151,Z 1173.449,A 0.000,B 0.000,C 90.000,E1 116.744} C_DIS
LIN {X -0.128,Y -706.637,Z 1173.444,A 0.000,B 0.000,C 90.000,E1 115.848} C_DIS
LIN {X -0.186,Y -706.750,Z 1173.440,A 0.000,B 0.000,C 90.000,E1 115.155} C_DIS
LIN {X 0.402,Y -706.550,Z 1173.437,A 0.000,B 0.000,C 90.000,E1 114.643} C_DIS
LIN {X -0.241,Y -706.301,Z 1173.436,A 0.000,B 0.000,C 90.000,E1 114.463} C_DIS
LIN {X 0.342,Y -705.363,Z 1173.433,A 0.000,B 0.000,C 90.000,E1 113.951} C_DIS
LIN {X -0.299,Y -704.496,Z 1173.432,A 0.000,B 0.000,C 90.000,E1 113.770} C_DIS
LIN {X 0.268,Y -702.338,Z 1173.429,A 0.000,B 0.000,C 90.000,E1 113.259} C_DIS
LIN {X 0.130,Y -701.439,Z 1173.429,A 0.000,B 0.000,C 90.000,E1 113.153} C_DIS
LIN {X 0.062,Y -696.700,Z 1173.426,A 0.000,B 0.000,C 90.000,E1 112.695} C_DIS
LIN {X -0.052,Y -695.049,Z 1173.426,A 0.000,B 0.000,C 90.000,E1 112.589} C_DIS
LIN {X 0.308,Y -692.591,Z 1173.425,A 0.000,B 0.000,C 90.000,E1 112.461} C_DIS
LIN {X 0.051,Y -686.049,Z 1173.424,A 0.000,B 0.000,C 90.000,E1 112.280} C_DIS
LIN {X -0.198,Y -685.117,Z 1173.424,A 0.000,B 0.000,C 90.000,E1 112.280} C_DIS
LIN {X -0.142,Y -683.588,Z 1173.424,A 0.000,B 0.000,C 90.000,E1 112.259} C_DIS
LIN {X 0.186,Y -677.511,Z 1173.423,A 0.000,B 0.000,C 90.000,E1 112.206} C_DIS
LIN {X 0.117,Y -605.226,Z 1173.423,A 0.000,B 0.000,C 90.000,E1 112.206} C_DIS
LIN {X -0.184,Y -600.245,Z 1173.422,A 0.000,B 0.000,C 90.000,E1 111.897} C_DIS
LIN {X -0.274,Y -596.099,Z 1173.420,A 0.000,B 0.000,C 90.000,E1 111.589} C_DIS
LIN {X 0.099,Y -585.667,Z 1173.415,A 0.000,B 0.000,C 90.000,E1 110.663} C_DIS
LIN {X -0.240,Y -574.347,Z 1173.410,A 0.000,B 0.000,C 90.000,E1 109.758} C_DIS
LIN {X 0.326,Y -566.705,Z 1173.407,A 0.000,B 0.000,C 90.000,E1 109.141} C_DIS
LIN {X 0.310,Y -556.120,Z 1173.403,A 0.000,B 0.000,C 90.000,E1 108.417} C_DIS
LIN {X 0.198,Y -551.892,Z 1173.401,A 0.000,B 0.000,C 90.000,E1 108.055} C_DIS
LIN {X -0.208,Y -550.631,Z 1173.399,A 0.000,B 0.000,C 90.000,E1 107.873} C_DIS
LIN {X 0.094,Y -550.107,Z 1173.397,A 0.000,B 0.000,C 90.000,E1 107.457} C_DIS
LIN {X 0.128,Y -550.664,Z 1173.391,A 0.000,B 0.000,C 90.000,E1 106.441} C_DIS
LIN {X 0.171,Y -551.639,Z 1173.385,A 0.000,B 0.000,C 90.000,E1 105.315} C_DIS
LIN {X 0.064,Y -553.177,Z 1173.376,A 0.000,B 0.000,C 90.000,E1 103.647} C_DIS
LIN {X -0.151,Y -554.950,Z 1173.365,A 0.000,B 0.000,C 90.000,E1 101.715} C_DIS
LIN {X 0.221,Y -556.965,Z 1173.354,A 0.000,B 0.000,C 90.000,E1 99.726} C_DIS
LIN {X -0.103,Y -558.875,Z 1173.343,A 0.000,B 0.000,C 90.000,E1 97.814} C_DIS
LIN {X -0.249,Y -559.762,Z 1173.337,A 0.000,B 0.000,C 90.000,E1 96.720} C_DIS
LIN {X -0.244,Y -560.802,Z 1173.330,A 0.000,B 0.000,C 90.000,E1 95.334} C_DIS
LIN {X 0.033,Y -562.290,Z 1173.317,A 0.000,B 0.000,C 90.000,E1 93.094} C_DIS
LIN {X 0.196,Y -563.734,Z 1173.307,A 0.000,B 0.000,C 90.000,E1 91.146} C_DIS
LIN {X 0.059,Y -564.604,Z 1173.300,A 0.000,B 0.000,C 90.000,E1 90.057} C_DIS
LIN {X 0.047,Y -565.553,Z 1173.293,A 0.000,B 0.000,C 90.000,E1 88.682} C_DIS
LIN {X 0.175,Y -566.632,Z 1173.284,A 0.000,B 0.000,C 90.000,E1 87.020} C_DIS
LIN {X -0.052,Y -567.842,Z 1173.273,A 0.000,B 0.000,C 90.000,E1 85.122} C_DIS
LIN {X 0.151,Y -568.976,Z 1173.264,A 0.000,B 0.000,C 90.000,E1 83.457} C_DIS
LIN {X -0.247,Y -569.889,Z 1173.256,A 0.000,B 0.000,C 90.000,E1 82.129} C_DIS
LIN {X 0.019,Y -570.659,Z 1173.249,A 0.000,B 0.000,C 90.000,E1 80.735} C_DIS
LIN {X -0.068,Y -571.526,Z 1173.240,A 0.000,B 0.000,C 90.000,E1 79.106} C_DIS
LIN {X -0.026,Y -572.374,Z 1173.230,A 0.000,B 0.000,C 90.000,E1 77.465} C_DIS
LIN {X -0.192,Y -573.352,Z 1173.220,A 0.000,B 0.000,C 90.000,E1 75.574} C_DIS
LIN {X -0.175,Y -573.975,Z 1173.212,A 0.000,B 0.000,C 90.000,E1 74.212} C_DIS
LIN {X -0.162,Y -575.096,Z 1173.202,A 0.000,B 0.000,C 90.000,E1 72.308} C_DIS
LIN {X -0.312,Y -576.712,Z 1173.188,A 0.000,B 0.000,C 90.000,E1 69.880} C_DIS
LIN {X 0.006,Y -578.743,Z 1173.175,A 0.000,B 0.000,C 90.000,E1 67.411} C_DIS
LIN {X 0.115,Y -580.106,Z 1173.167,A 0.000,B 0.000,C 90.000,E1 66.049} C_DIS
LIN {X 0.207,Y -581.886,Z 1173.157,A 0.000,B 0.000,C 90.000,E1 64.152} C_DIS
LIN {X 0.078,Y -583.645,Z 1173.146,A 0.000,B 0.000,C 90.000,E1 62.281} C_DIS
LIN {X 0.113,Y -585.156,Z 1173.137,A 0.000,B 0.000,C 90.000,E1 60.667} C_DIS
LIN {X 0.071,Y -586.337,Z 1173.130,A 0.000,B 0.000,C 90.000,E1 59.331} C_DIS
LIN {X 0.052,Y -587.375,Z 1173.122,A 0.000,B 0.000,C 90.000,E1 57.995} C_DIS
LIN {X -0.258,Y -588.501,Z 1173.113,A 0.000,B 0.000,C 90.000,E1 56.421} C_DIS
LIN {X 0.005,Y -589.031,Z 1173.109,A 0.000,B 0.000,C 90.000,E1 55.595} C_DIS
LIN {X -0.009,Y -589.780,Z 1173.103,A 0.000,B 0.000,C 90.000,E1 54.529} C_DIS
LIN {X 0.263,Y -590.947,Z 1173.093,A 0.000,B 0.000,C 90.000,E1 52.637} C_DIS
LIN {X -0.240,Y -591.886,Z 1173.084,A 0.000,B 0.000,C 90.000,E1 51.090} C_DIS
LIN {X -0.065,Y -592.372,Z 1173.079,A 0.000,B 0.000,C 90.000,E1 50.275} C_DIS
LIN {X 0.082,Y -592.825,Z 1173.072,A 0.000,B 0.000,C 90.000,E1 48.933} C_DIS
LIN {X 0.020,Y -593.128,Z 1173.066,A 0.000,B 0.000,C 90.000,E1 47.877} C_DIS
LIN {X 0.124,Y -593.344,Z 1173.059,A 0.000,B 0.000,C 90.000,E1 46.539} C_DIS
LIN {X 0.038,Y -593.276,Z 1173.053,A 0.000,B 0.000,C 90.000,E1 45.486} C_DIS
LIN {X -0.046,Y -593.029,Z 1173.047,A 0.000,B 0.000,C 90.000,E1 44.433} C_DIS
LIN {X 0.097,Y -592.743,Z 1173.042,A 0.000,B 0.000,C 90.000,E1 43.623} C_DIS
LIN {X -0.172,Y -592.309,Z 1173.038,A 0.000,B 0.000,C 90.000,E1 42.852} C_DIS
LIN {X -0.085,Y -591.462,Z 1173.031,A 0.000,B 0.000,C 90.000,E1 41.515} C_DIS
LIN {X 0.079,Y -590.853,Z 1173.026,A 0.000,B 0.000,C 90.000,E1 40.701} C_DIS
LIN {X 0.195,Y -589.486,Z 1173.019,A 0.000,B 0.000,C 90.000,E1 39.358} C_DIS
LIN {X -0.116,Y -588.549,Z 1173.014,A 0.000,B 0.000,C 90.000,E1 38.588} C_DIS
LIN {X 0.049,Y -586.728,Z 1173.007,A 0.000,B 0.000,C 90.000,E1 37.237} C_DIS
LIN {X 0.001,Y -584.907,Z 1173.001,A 0.000,B 0.000,C 90.000,E1 36.171} C_DIS
LIN {X -0.254,Y -583.259,Z 1172.997,A 0.000,B 0.000,C 90.000,E1 35.391} C_DIS
LIN {X 0.281,Y -581.518,Z 1172.992,A 0.000,B 0.000,C 90.000,E1 34.532} C_DIS
LIN {X -0.341,Y -579.327,Z 1172.988,A 0.000,B 0.000,C 90.000,E1 33.785} C_DIS
LIN {X -0.178,Y -576.889,Z 1172.983,A 0.000,B 0.000,C 90.000,E1 32.959} C_DIS
LIN {X -0.045,Y -574.089,Z 1172.979,A 0.000,B 0.000,C 90.000,E1 32.133} C_DIS
LIN {X -0.245,Y -570.847,Z 1172.974,A 0.000,B 0.000,C 90.000,E1 31.337} C_DIS
LIN {X 0.103,Y -567.867,Z 1172.970,A 0.000,B 0.000,C 90.000,E1 30.620} C_DIS
LIN {X 0.029,Y -565.293,Z 1172.967,A 0.000,B 0.000,C 90.000,E1 30.079} C_DIS
LIN {X -0.068,Y -562.509,Z 1172.964,A 0.000,B 0.000,C 90.000,E1 29.539} C_DIS
LIN {X 0.098,Y -557.908,Z 1172.959,A 0.000,B 0.000,C 90.000,E1 28.693} C_DIS
LIN {X -0.165,Y -553.865,Z 1172.956,A 0.000,B 0.000,C 90.000,E1 28.025} C_DIS
LIN {X 0.019,Y -549.504,Z 1172.952,A 0.000,B 0.000,C 90.000,E1 27.308} C_DIS
LIN {X -0.085,Y -544.700,Z 1172.948,A 0.000,B 0.000,C 90.000,E1 26.616} C_DIS
LIN {X 0.030,Y -541.650,Z 1172.946,A 0.000,B 0.000,C 90.000,E1 26.181} C_DIS
LIN {X 0.231,Y -537.325,Z 1172.942,A 0.000,B 0.000,C 90.000,E1 25.591} C_DIS
LIN {X -0.027,Y -534.108,Z 1172.940,A 0.000,B 0.000,C 90.000,E1 25.207} C_DIS
LIN {X 0.135,Y -525.782,Z 1172.935,A 0.000,B 0.000,C 90.000,E1 24.207} C_DIS
LIN {X 0.002,Y -519.467,Z 1172.931,A 0.000,B 0.000,C 90.000,E1 23.515} C_DIS
LIN {X -0.132,Y -512.857,Z 1172.927,A 0.000,B 0.000,C 90.000,E1 22.823} C_DIS
LIN {X 0.120,Y -504.785,Z 1172.922,A 0.000,B 0.000,C 90.000,E1 21.972} C_DIS
LIN {X 0.271,Y -497.827,Z 1172.918,A 0.000,B 0.000,C 90.000,E1 21.280} C_DIS
LIN {X 0.007,Y -487.817,Z 1172.913,A 0.000,B 0.000,C 90.000,E1 20.375} C_DIS
LIN {X 0.087,Y -476.214,Z 1172.907,A 0.000,B 0.000,C 90.000,E1 19.322} C_DIS
LIN {X 0.222,Y -470.357,Z 1172.905,A 0.000,B 0.000,C 90.000,E1 18.779} C_DIS
LIN {X -0.146,Y -461.661,Z 1172.900,A 0.000,B 0.000,C 90.000,E1 18.055} C_DIS
LIN {X 0.073,Y -444.460,Z 1172.891,A 0.000,B 0.000,C 90.000,E1 16.441} C_DIS
LIN {X 0.151,Y -427.369,Z 1172.882,A 0.000,B 0.000,C 90.000,E1 14.717} C_DIS
LIN {X -0.022,Y -414.923,Z 1172.874,A 0.000,B 0.000,C 90.000,E1 13.355} C_DIS
LIN {X 0.002,Y -405.478,Z 1172.868,A 0.000,B 0.000,C 90.000,E1 12.187} C_DIS
LIN {X -0.112,Y -399.322,Z 1172.863,A 0.000,B 0.000,C 90.000,E1 11.366} C_DIS
LIN {X -0.095,Y -395.897,Z 1172.860,A 0.000,B 0.000,C 90.000,E1 10.838} C_DIS
LIN {X -0.103,Y -393.844,Z 1172.858,A 0.000,B 0.000,C 90.000,E1 10.423} C_DIS
LIN {X -0.128,Y -393.340,Z 1172.857,A 0.000,B 0.000,C 90.000,E1 10.254} C_DIS
LIN {X 0.167,Y -392.767,Z 1172.855,A 0.000,B 0.000,C 90.000,E1 9.962} C_DIS
LIN {X 0.129,Y -392.771,Z 1172.855,A 0.000,B 0.000,C 90.000,E1 9.962} C_DIS
LIN {X 0.179,Y -393.286,Z 1172.853,A 0.000,B 0.000,C 90.000,E1 9.500} C_DIS
LIN {X 0.100,Y -395.035,Z 1172.849,A 0.000,B 0.000,C 90.000,E1 8.803} C_DIS
LIN {X -0.008,Y -398.192,Z 1172.844,A 0.000,B 0.000,C 90.000,E1 7.936} C_DIS
LIN {X -0.083,Y -402.151,Z 1172.839,A 0.000,B 0.000,C 90.000,E1 7.068} C_DIS
LIN {X -0.193,Y -407.162,Z 1172.835,A 0.000,B 0.000,C 90.000,E1 6.372} C_DIS
LIN {X -0.163,Y -412.199,Z 1172.833,A 0.000,B 0.000,C 90.000,E1 5.910} C_DIS
LIN {X -0.024,Y -427.825,Z 1172.826,A 0.000,B 0.000,C 90.000,E1 4.702} C_DIS
LIN {X 0.098,Y -451.987,Z 1172.816,A 0.000,B 0.000,C 90.000,E1 2.922} C_DIS
LIN {X -0.159,Y -466.189,Z 1172.811,A 0.000,B 0.000,C 90.000,E1 1.949} C_DIS
LIN {X -0.117,Y -474.105,Z 1172.808,A 0.000,B 0.000,C 90.000,E1 1.375} C_DIS
LIN {X -0.149,Y -480.366,Z 1172.805,A 0.000,B 0.000,C 90.000,E1 0.917} C_DIS
LIN {X 0.208,Y -486.502,Z 1172.802,A 0.000,B 0.000,C 90.000,E1 0.401} C_DIS
LIN {X 0.060,Y -491.022,Z 1172.800,A 0.000,B 0.000,C 90.000,E1 0.057} C_DIS
LIN {X 0.022,Y -497.205,Z 1172.797,A 0.000,B 0.000,C 90.000,E1 359.542} C_DIS
LIN {X -0.155,Y -504.141,Z 1172.794,A 0.000,B 0.000,C 90.000,E1 358.912} C_DIS
LIN {X -0.174,Y -510.823,Z 1172.790,A 0.000,B 0.000,C 90.000,E1 358.224} C_DIS
LIN {X 0.079,Y -517.174,Z 1172.786,A 0.000,B 0.000,C 90.000,E1 357.478} C_DIS
LIN {X -0.080,Y -523.053,Z 1172.782,A 0.000,B 0.000,C 90.000,E1 356.788} C_DIS
LIN {X 0.071,Y -528.490,Z 1172.778,A 0.000,B 0.000,C 90.000,E1 356.045} C_DIS
LIN {X 0.051,Y -532.529,Z 1172.775,A 0.000,B 0.000,C 90.000,E1 355.469} C_DIS
LIN {X -0.212,Y -537.078,Z 1172.771,A 0.000,B 0.000,C 90.000,E1 354.780} C_DIS
LIN {X 0.101,Y -541.143,Z 1172.767,A 0.000,B 0.000,C 90.000,E1 354.033} C_DIS
LIN {X 0.173,Y -544.130,Z 1172.764,A 0.000,B 0.000,C 90.000,E1 353.457} C_DIS
LIN {X 0.072,Y -547.496,Z 1172.760,A 0.000,B 0.000,C 90.000,E1 352.761} C_DIS
LIN {X 0.190,Y -550.016,Z 1172.757,A 0.000,B 0.000,C 90.000,E1 352.186} C_DIS
LIN {X -0.143,Y -552.337,Z 1172.754,A 0.000,B 0.000,C 90.000,E1 351.659} C_DIS
LIN {X 0.124,Y -555.465,Z 1172.749,A 0.000,B 0.000,C 90.000,E1 350.792} C_DIS
LIN {X -0.261,Y -557.389,Z 1172.746,A 0.000,B 0.000,C 90.000,E1 350.274} C_DIS
LIN {X 0.153,Y -559.998,Z 1172.741,A 0.000,B 0.000,C 90.000,E1 349.398} C_DIS
LIN {X 0.205,Y -563.147,Z 1172.735,A 0.000,B 0.000,C 90.000,E1 348.285} C_DIS
LIN {X 0.137,Y -565.343,Z 1172.730,A 0.000,B 0.000,C 90.000,E1 347.465} C_DIS
LIN {X 0.090,Y -567.492,Z 1172.726,A 0.000,B 0.000,C 90.000,E1 346.645} C_DIS
LIN {X 0.190,Y -571.352,Z 1172.717,A 0.000,B 0.000,C 90.000,E1 344.991} C_DIS
LIN {X -0.017,Y -573.777,Z 1172.711,A 0.000,B 0.000,C 90.000,E1 343.921} C_DIS
LIN {X -0.193,Y -577.201,Z 1172.702,A 0.000,B 0.000,C 90.000,E1 342.308} C_DIS
LIN {X 0.227,Y -579.775,Z 1172.694,A 0.000,B 0.000,C 90.000,E1 340.913} C_DIS
LIN {X -0.245,Y -581.597,Z 1172.688,A 0.000,B 0.000,C 90.000,E1 339.880} C_DIS
LIN {X 0.055,Y -583.236,Z 1172.682,A 0.000,B 0.000,C 90.000,E1 338.773} C_DIS
LIN {X 0.248,Y -584.832,Z 1172.675,A 0.000,B 0.000,C 90.000,E1 337.411} C_DIS
LIN {X 0.176,Y -585.443,Z 1172.670,A 0.000,B 0.000,C 90.000,E1 336.613} C_DIS
LIN {X 0.220,Y -585.850,Z 1172.664,A 0.000,B 0.000,C 90.000,E1 335.537} C_DIS
LIN {X -0.137,Y -585.670,Z 1172.660,A 0.000,B 0.000,C 90.000,E1 334.768} C_DIS
LIN {X 0.035,Y -585.255,Z 1172.655,A 0.000,B 0.000,C 90.000,E1 333.948} C_DIS
LIN {X 0.319,Y -584.829,Z 1172.652,A 0.000,B 0.000,C 90.000,E1 333.384} C_DIS
LIN {X -0.049,Y -583.769,Z 1172.648,A 0.000,B 0.000,C 90.000,E1 332.615} C_DIS
LIN {X 0.229,Y -581.908,Z 1172.642,A 0.000,B 0.000,C 90.000,E1 331.513} C_DIS
LIN {X 0.108,Y -580.006,Z 1172.637,A 0.000,B 0.000,C 90.000,E1 330.717} C_DIS
LIN {X -0.172,Y -578.567,Z 1172.634,A 0.000,B 0.000,C 90.000,E1 330.205} C_DIS
LIN {X -0.176,Y -576.949,Z 1172.631,A 0.000,B 0.000,C 90.000,E1 329.665} C_DIS
LIN {X -0.186,Y -574.898,Z 1172.628,A 0.000,B 0.000,C 90.000,E1 329.125} C_DIS
LIN {X 0.147,Y -573.777,Z 1172.627,A 0.000,B 0.000,C 90.000,E1 328.820} C_DIS
LIN {X 0.234,Y -569.549,Z 1172.622,A 0.000,B 0.000,C 90.000,E1 327.995} C_DIS
LIN {X 0.169,Y -566.365,Z 1172.619,A 0.000,B 0.000,C 90.000,E1 327.454} C_DIS
LIN {X 0.330,Y -561.107,Z 1172.615,A 0.000,B 0.000,C 90.000,E1 326.628} C_DIS
LIN {X 0.202,Y -557.105,Z 1172.612,A 0.000,B 0.000,C 90.000,E1 326.087} C_DIS
LIN {X 0.165,Y -553.882,Z 1172.609,A 0.000,B 0.000,C 90.000,E1 325.674} C_DIS
LIN {X 0.172,Y -548.232,Z 1172.606,A 0.000,B 0.000,C 90.000,E1 324.975} C_DIS
LIN {X -0.016,Y -540.812,Z 1172.601,A 0.000,B 0.000,C 90.000,E1 324.149} C_DIS
LIN {X -0.161,Y -528.171,Z 1172.593,A 0.000,B 0.000,C 90.000,E1 322.763} C_DIS
LIN {X -0.126,Y -524.759,Z 1172.591,A 0.000,B 0.000,C 90.000,E1 322.351} C_DIS
LIN {X 0.009,Y -521.098,Z 1172.588,A 0.000,B 0.000,C 90.000,E1 321.823} C_DIS
LIN {X 0.102,Y -518.744,Z 1172.586,A 0.000,B 0.000,C 90.000,E1 321.376} C_DIS
LIN {X -0.013,Y -516.913,Z 1172.582,A 0.000,B 0.000,C 90.000,E1 320.803} C_DIS
LIN {X -0.220,Y -516.075,Z 1172.578,A 0.000,B 0.000,C 90.000,E1 320.070} C_DIS
LIN {X -0.028,Y -516.055,Z 1172.575,A 0.000,B 0.000,C 90.000,E1 319.461} C_DIS
LIN {X 0.093,Y -517.083,Z 1172.563,A 0.000,B 0.000,C 90.000,E1 317.391} C_DIS
LIN {X -0.064,Y -518.085,Z 1172.554,A 0.000,B 0.000,C 90.000,E1 315.648} C_DIS
LIN {X -0.041,Y -518.732,Z 1172.547,A 0.000,B 0.000,C 90.000,E1 314.474} C_DIS
LIN {X -0.076,Y -519.557,Z 1172.539,A 0.000,B 0.000,C 90.000,E1 313.014} C_DIS
LIN {X -0.247,Y -520.812,Z 1172.528,A 0.000,B 0.000,C 90.000,E1 310.987} C_DIS
LIN {X 0.156,Y -521.698,Z 1172.520,A 0.000,B 0.000,C 90.000,E1 309.483} C_DIS
LIN {X 0.155,Y -522.988,Z 1172.508,A 0.000,B 0.000,C 90.000,E1 307.443} C_DIS
LIN {X -0.052,Y -523.766,Z 1172.500,A 0.000,B 0.000,C 90.000,E1 306.011} C_DIS
LIN {X 0.160,Y -525.273,Z 1172.486,A 0.000,B 0.000,C 90.000,E1 303.372} C_DIS
LIN {X 0.158,Y -525.992,Z 1172.479,A 0.000,B 0.000,C 90.000,E1 302.212} C_DIS
LIN {X 0.255,Y -526.902,Z 1172.469,A 0.000,B 0.000,C 90.000,E1 300.463} C_DIS
LIN {X 0.045,Y -527.271,Z 1172.465,A 0.000,B 0.000,C 90.000,E1 299.617} C_DIS
LIN {X 0.201,Y -527.760,Z 1172.457,A 0.000,B 0.000,C 90.000,E1 298.153} C_DIS
LIN {X 0.032,Y -528.076,Z 1172.447,A 0.000,B 0.000,C 90.000,E1 296.437} C_DIS
LIN {X 0.006,Y -528.244,Z 1172.441,A 0.000,B 0.000,C 90.000,E1 295.283} C_DIS
LIN {X 0.151,Y -528.255,Z 1172.432,A 0.000,B 0.000,C 90.000,E1 293.823} C_DIS
LIN {X 0.053,Y -528.127,Z 1172.423,A 0.000,B 0.000,C 90.000,E1 292.099} C_DIS
LIN {X -0.037,Y -527.845,Z 1172.413,A 0.000,B 0.000,C 90.000,E1 290.375} C_DIS
LIN {X -0.147,Y -527.393,Z 1172.402,A 0.000,B 0.000,C 90.000,E1 288.362} C_DIS
LIN {X -0.290,Y -527.003,Z 1172.396,A 0.000,B 0.000,C 90.000,E1 287.221} C_DIS
LIN {X 0.065,Y -526.596,Z 1172.389,A 0.000,B 0.000,C 90.000,E1 286.024} C_DIS
LIN {X -0.085,Y -525.857,Z 1172.381,A 0.000,B 0.000,C 90.000,E1 284.592} C_DIS
LIN {X -0.032,Y -525.282,Z 1172.376,A 0.000,B 0.000,C 90.000,E1 283.716} C_DIS
LIN {X 0.189,Y -524.149,Z 1172.367,A 0.000,B 0.000,C 90.000,E1 281.951} C_DIS
LIN {X -0.266,Y -523.444,Z 1172.360,A 0.000,B 0.000,C 90.000,E1 280.838} C_DIS
LIN {X 0.231,Y -522.158,Z 1172.349,A 0.000,B 0.000,C 90.000,E1 278.746} C_DIS
LIN {X 0.101,Y -521.069,Z 1172.339,A 0.000,B 0.000,C 90.000,E1 277.011} C_DIS
LIN {X -0.124,Y -519.842,Z 1172.328,A 0.000,B 0.000,C 90.000,E1 274.992} C_DIS
LIN {X 0.019,Y -518.693,Z 1172.315,A 0.000,B 0.000,C 90.000,E1 272.636} C_DIS
LIN {X 0.136,Y -517.705,Z 1172.303,A 0.000,B 0.000,C 90.000,E1 270.573} C_DIS
LIN {X -0.234,Y -516.931,Z 1172.294,A 0.000,B 0.000,C 90.000,E1 268.854} C_DIS
LIN {X -0.028,Y -516.290,Z 1172.285,A 0.000,B 0.000,C 90.000,E1 267.364} C_DIS
LIN {X 0.233,Y -515.582,Z 1172.279,A 0.000,B 0.000,C 90.000,E1 266.159} C_DIS
LIN {X -0.074,Y -514.454,Z 1172.271,A 0.000,B 0.000,C 90.000,E1 264.723} C_DIS
LIN {X 0.031,Y -512.661,Z 1172.259,A 0.000,B 0.000,C 90.000,E1 262.648} C_DIS
LIN {X -0.172,Y -511.529,Z 1172.253,A 0.000,B 0.000,C 90.000,E1 261.489} C_DIS
LIN {X -0.039,Y -509.299,Z 1172.240,A 0.000,B 0.000,C 90.000,E1 259.106} C_DIS
LIN {X -0.289,Y -507.792,Z 1172.230,A 0.000,B 0.000,C 90.000,E1 257.353} C_DIS
LIN {X 0.094,Y -506.058,Z 1172.218,A 0.000,B 0.000,C 90.000,E1 255.227} C_DIS
LIN {X -0.001,Y -504.509,Z 1172.208,A 0.000,B 0.000,C 90.000,E1 253.449} C_DIS
LIN {X 0.076,Y -502.719,Z 1172.197,A 0.000,B 0.000,C 90.000,E1 251.348} C_DIS
LIN {X -0.111,Y -501.034,Z 1172.187,A 0.000,B 0.000,C 90.000,E1 249.571} C_DIS
LIN {X 0.067,Y -499.627,Z 1172.178,A 0.000,B 0.000,C 90.000,E1 248.050} C_DIS
LIN {X 0.131,Y -498.175,Z 1172.170,A 0.000,B 0.000,C 90.000,E1 246.538} C_DIS
LIN {X 0.233,Y -496.023,Z 1172.160,A 0.000,B 0.000,C 90.000,E1 244.717} C_DIS
LIN {X -0.071,Y -494.927,Z 1172.155,A 0.000,B 0.000,C 90.000,E1 243.845} C_DIS
LIN {X -0.059,Y -492.487,Z 1172.145,A 0.000,B 0.000,C 90.000,E1 242.025} C_DIS
LIN {X -0.100,Y -490.014,Z 1172.134,A 0.000,B 0.000,C 90.000,E1 240.205} C_DIS
LIN {X 0.046,Y -487.889,Z 1172.126,A 0.000,B 0.000,C 90.000,E1 238.663} C_DIS
LIN {X -0.027,Y -485.241,Z 1172.116,A 0.000,B 0.000,C 90.000,E1 236.834} C_DIS
LIN {X 0.128,Y -481.710,Z 1172.102,A 0.000,B 0.000,C 90.000,E1 234.356} C_DIS
LIN {X 0.239,Y -480.422,Z 1172.097,A 0.000,B 0.000,C 90.000,E1 233.417} C_DIS
LIN {X -0.245,Y -477.747,Z 1172.087,A 0.000,B 0.000,C 90.000,E1 231.618} C_DIS
LIN {X -0.190,Y -475.198,Z 1172.076,A 0.000,B 0.000,C 90.000,E1 229.747} C_DIS
LIN {X 0.027,Y -473.160,Z 1172.068,A 0.000,B 0.000,C 90.000,E1 228.162} C_DIS
LIN {X -0.156,Y -470.592,Z 1172.059,A 0.000,B 0.000,C 90.000,E1 226.620} C_DIS
LIN {X 0.036,Y -465.866,Z 1172.040,A 0.000,B 0.000,C 90.000,E1 223.137} C_DIS
LIN {X -0.081,Y -462.813,Z 1172.017,A 0.000,B 0.000,C 90.000,E1 219.036} C_DIS
LIN {X 0.082,Y -462.192,Z 1172.006,A 0.000,B 0.000,C 90.000,E1 217.111} C_DIS
LIN {X -0.142,Y -461.553,Z 1171.990,A 0.000,B 0.000,C 90.000,E1 214.278} C_DIS
LIN {X 0.108,Y -461.624,Z 1171.980,A 0.000,B 0.000,C 90.000,E1 212.339} C_DIS
LIN {X -0.100,Y -463.606,Z 1171.960,A 0.000,B 0.000,C 90.000,E1 208.871} C_DIS
LIN {X -0.148,Y -466.080,Z 1171.945,A 0.000,B 0.000,C 90.000,E1 206.027} C_DIS
LIN {X 0.197,Y -471.460,Z 1171.924,A 0.000,B 0.000,C 90.000,E1 202.206} C_DIS
LIN {X 0.180,Y -476.996,Z 1171.908,A 0.000,B 0.000,C 90.000,E1 199.396} C_DIS
LIN {X 0.054,Y -484.941,Z 1171.891,A 0.000,B 0.000,C 90.000,E1 196.315} C_DIS
LIN {X -0.203,Y -493.348,Z 1171.875,A 0.000,B 0.000,C 90.000,E1 193.592} C_DIS
LIN {X -0.251,Y -500.338,Z 1171.864,A 0.000,B 0.000,C 90.000,E1 191.478} C_DIS
LIN {X -0.221,Y -507.468,Z 1171.852,A 0.000,B 0.000,C 90.000,E1 189.378} C_DIS
LIN {X -0.135,Y -513.909,Z 1171.842,A 0.000,B 0.000,C 90.000,E1 187.587} C_DIS
LIN {X 0.121,Y -519.154,Z 1171.834,A 0.000,B 0.000,C 90.000,E1 186.087} C_DIS
LIN {X -0.143,Y -526.388,Z 1171.823,A 0.000,B 0.000,C 90.000,E1 184.073} C_DIS
LIN {X -0.233,Y -531.560,Z 1171.815,A 0.000,B 0.000,C 90.000,E1 182.636} C_DIS
LIN {X -0.263,Y -536.603,Z 1171.807,A 0.000,B 0.000,C 90.000,E1 181.203} C_DIS
LIN {X -0.191,Y -542.790,Z 1171.797,A 0.000,B 0.000,C 90.000,E1 179.484} C_DIS
LIN {X -0.013,Y -547.894,Z 1171.789,A 0.000,B 0.000,C 90.000,E1 178.051} C_DIS
LIN {X 0.265,Y -552.912,Z 1171.781,A 0.000,B 0.000,C 90.000,E1 176.617} C_DIS
LIN {X 0.262,Y -559.931,Z 1171.771,A 0.000,B 0.000,C 90.000,E1 174.666} C_DIS
LIN {X 0.288,Y -564.910,Z 1171.763,A 0.000,B 0.000,C 90.000,E1 173.280} C_DIS
LIN {X -0.157,Y -569.820,Z 1171.755,A 0.000,B 0.000,C 90.000,E1 171.951} C_DIS
LIN {X 0.237,Y -575.658,Z 1171.746,A 0.000,B 0.000,C 90.000,E1 170.274} C_DIS
LIN {X 0.295,Y -578.569,Z 1171.742,A 0.000,B 0.000,C 90.000,E1 169.454} C_DIS
LIN {X -0.175,Y -584.241,Z 1171.733,A 0.000,B 0.000,C 90.000,E1 167.881} C_DIS
LIN {X 0.293,Y -589.824,Z 1171.724,A 0.000,B 0.000,C 90.000,E1 166.228} C_DIS
LIN {X 0.316,Y -595.181,Z 1171.715,A 0.000,B 0.000,C 90.000,E1 164.629} C_DIS
LIN {X -0.136,Y -600.469,Z 1171.706,A 0.000,B 0.000,C 90.000,E1 163.087} C_DIS
LIN {X -0.045,Y -604.681,Z 1171.699,A 0.000,B 0.000,C 90.000,E1 161.764} C_DIS
LIN {X 0.318,Y -608.679,Z 1171.691,A 0.000,B 0.000,C 90.000,E1 160.423} C_DIS
LIN {X -0.079,Y -613.336,Z 1171.683,A 0.000,B 0.000,C 90.000,E1 158.901} C_DIS
LIN {X 0.118,Y -616.309,Z 1171.677,A 0.000,B 0.000,C 90.000,E1 157.847} C_DIS
LIN {X 0.075,Y -621.408,Z 1171.667,A 0.000,B 0.000,C 90.000,E1 156.049} C_DIS
LIN {X -0.189,Y -624.920,Z 1171.660,A 0.000,B 0.000,C 90.000,E1 154.793} C_DIS
LIN {X -0.084,Y -629.647,Z 1171.650,A 0.000,B 0.000,C 90.000,E1 152.999} C_DIS
LIN {X 0.025,Y -632.245,Z 1171.644,A 0.000,B 0.000,C 90.000,E1 151.975} C_DIS
LIN {X -0.048,Y -635.385,Z 1171.637,A 0.000,B 0.000,C 90.000,E1 150.717} C_DIS
LIN {X -0.061,Y -638.353,Z 1171.630,A 0.000,B 0.000,C 90.000,E1 149.459} C_DIS
LIN {X -0.030,Y -641.087,Z 1171.623,A 0.000,B 0.000,C 90.000,E1 148.201} C_DIS
LIN {X -0.023,Y -643.200,Z 1171.618,A 0.000,B 0.000,C 90.000,E1 147.199} C_DIS
LIN {X -0.126,Y -645.556,Z 1171.611,A 0.000,B 0.000,C 90.000,E1 145.960} C_DIS
LIN {X 0.134,Y -648.644,Z 1171.601,A 0.000,B 0.000,C 90.000,E1 144.196} C_DIS
LIN {X -0.020,Y -650.831,Z 1171.594,A 0.000,B 0.000,C 90.000,E1 142.970} C_DIS
LIN {X 0.397,Y -652.130,Z 1171.590,A 0.000,B 0.000,C 90.000,E1 142.190} C_DIS
LIN {X 0.240,Y -654.709,Z 1171.582,A 0.000,B 0.000,C 90.000,E1 140.723} C_DIS
LIN {X 0.085,Y -658.101,Z 1171.572,A 0.000,B 0.000,C 90.000,E1 139.013} C_DIS
LIN {X -0.014,Y -660.687,Z 1171.566,A 0.000,B 0.000,C 90.000,E1 137.796} C_DIS
LIN {X 0.352,Y -664.238,Z 1171.556,A 0.000,B 0.000,C 90.000,E1 136.053} C_DIS
LIN {X 0.338,Y -668.934,Z 1171.544,A 0.000,B 0.000,C 90.000,E1 133.866} C_DIS
LIN {X -0.034,Y -673.516,Z 1171.533,A 0.000,B 0.000,C 90.000,E1 131.962} C_DIS
LIN {X -0.097,Y -679.914,Z 1171.518,A 0.000,B 0.000,C 90.000,E1 129.322} C_DIS
LIN {X 0.054,Y -684.662,Z 1171.508,A 0.000,B 0.000,C 90.000,E1 127.397} C_DIS
LIN {X 0.127,Y -688.204,Z 1171.500,A 0.000,B 0.000,C 90.000,E1 125.964} C_DIS
LIN {X -0.343,Y -691.150,Z 1171.493,A 0.000,B 0.000,C 90.000,E1 124.818} C_DIS
LIN {X -0.213,Y -693.889,Z 1171.487,A 0.000,B 0.000,C 90.000,E1 123.627} C_DIS
LIN {X 0.159,Y -696.523,Z 1171.480,A 0.000,B 0.000,C 90.000,E1 122.418} C_DIS
LIN {X 0.332,Y -698.473,Z 1171.475,A 0.000,B 0.000,C 90.000,E1 121.465} C_DIS
LIN {X 0.093,Y -701.169,Z 1171.467,A 0.000,B 0.000,C 90.000,E1 120.079} C_DIS
LIN {X -0.093,Y -703.598,Z 1171.459,A 0.000,B 0.000,C 90.000,E1 118.693} C_DIS
LIN {X 0.087,Y -705.392,Z 1171.453,A 0.000,B 0.000,C 90.000,E1 117.513} C_DIS
LIN {X 0.010,Y -706.121,Z 1171.449,A 0.000,B 0.000,C 90.000,E1 116.821} C_DIS
LIN {X -0.083,Y -706.611,Z 1171.444,A 0.000,B 0.000,C 90.000,E1 115.899} C_DIS
LIN {X -0.145,Y -706.743,Z 1171.440,A 0.000,B 0.000,C 90.000,E1 115.207} C_DIS
LIN {X -0.204,Y -706.416,Z 1171.436,A 0.000,B 0.000,C 90.000,E1 114.515} C_DIS
LIN {X 0.091,Y -705.470,Z 1171.434,A 0.000,B 0.000,C 90.000,E1 114.027} C_DIS
LIN {X -0.265,Y -704.750,Z 1171.432,A 0.000,B 0.000,C 90.000,E1 113.823} C_DIS
LIN {X 0.024,Y -702.632,Z 1171.430,A 0.000,B 0.000,C 90.000,E1 113.334} C_DIS
LIN {X 0.163,Y -701.890,Z 1171.429,A 0.000,B 0.000,C 90.000,E1 113.206} C_DIS
LIN {X -0.212,Y -697.299,Z 1171.426,A 0.000,B 0.000,C 90.000,E1 112.770} C_DIS
LIN {X -0.082,Y -695.917,Z 1171.426,A 0.000,B 0.000,C 90.000,E1 112.642} C_DIS
LIN {X 0.149,Y -693.860,Z 1171.425,A 0.000,B 0.000,C 90.000,E1 112.514} C_DIS
LIN {X -0.121,Y -685.592,Z 1171.424,A 0.000,B 0.000,C 90.000,E1 112.280} C_DIS
LIN {X -0.159,Y -683.919,Z 1171.424,A 0.000,B 0.000,C 90.000,E1 112.259} C_DIS
LIN {X 0.097,Y -677.105,Z 1171.423,A 0.000,B 0.000,C 90.000,E1 112.206} C_DIS
LIN {X 0.039,Y -605.040,Z 1171.423,A 0.000,B 0.000,C 90.000,E1 112.206} C_DIS
LIN {X 0.115,Y -599.126,Z 1171.421,A 0.000,B 0.000,C 90.000,E1 111.791} C_DIS
LIN {X 0.142,Y -594.952,Z 1171.419,A 0.000,B 0.000,C 90.000,E1 111.461} C_DIS
LIN {X -0.178,Y -583.990,Z 1171.414,A 0.000,B 0.000,C 90.000,E1 110.556} C_DIS
LIN {X 0.123,Y -574.151,Z 1171.410,A 0.000,B 0.000,C 90.000,E1 109.704} C_DIS
LIN {X 0.068,Y -568.292,Z 1171.407,A 0.000,B 0.000,C 90.000,E1 109.268} C_DIS
LIN {X -0.167,Y -558.889,Z 1171.404,A 0.000,B 0.000,C 90.000,E1 108.652} C_DIS
LIN {X 0.111,Y -555.861,Z 1171.402,A 0.000,B 0.000,C 90.000,E1 108.417} C_DIS
LIN {X -0.140,Y -552.172,Z 1171.401,A 0.000,B 0.000,C 90.000,E1 108.127} C_DIS
LIN {X -0.201,Y -550.527,Z 1171.399,A 0.000,B 0.000,C 90.000,E1 107.873} C_DIS
LIN {X -0.104,Y -550.126,Z 1171.398,A 0.000,B 0.000,C 90.000,E1 107.583} C_DIS
LIN {X -0.235,Y -550.051,Z 1171.397,A 0.000,B 0.000,C 90.000,E1 107.457} C_DIS
LIN {X -0.206,Y -550.684,Z 1171.391,A 0.000,B 0.000,C 90.000,E1 106.441} C_DIS
LIN {X -0.018,Y -551.652,Z 1171.385,A 0.000,B 0.000,C 90.000,E1 105.300} C_DIS
LIN {X -0.152,Y -553.405,Z 1171.374,A 0.000,B 0.000,C 90.000,E1 103.355} C_DIS
LIN {X 0.056,Y -554.954,Z 1171.365,A 0.000,B 0.000,C 90.000,E1 101.658} C_DIS
LIN {X -0.074,Y -557.205,Z 1171.352,A 0.000,B 0.000,C 90.000,E1 99.443} C_DIS
LIN {X 0.175,Y -559.073,Z 1171.342,A 0.000,B 0.000,C 90.000,E1 97.473} C_DIS
LIN {X 0.103,Y -559.911,Z 1171.335,A 0.000,B 0.000,C 90.000,E1 96.372} C_DIS
LIN {X 0.056,Y -560.945,Z 1171.328,A 0.000,B 0.000,C 90.000,E1 94.992} C_DIS
LIN {X -0.215,Y -562.456,Z 1171.316,A 0.000,B 0.000,C 90.000,E1 92.808} C_DIS
LIN {X -0.046,Y -563.888,Z 1171.305,A 0.000,B 0.000,C 90.000,E1 90.859} C_DIS
LIN {X -0.179,Y -564.746,Z 1171.299,A 0.000,B 0.000,C 90.000,E1 89.771} C_DIS
LIN {X 0.262,Y -565.510,Z 1171.293,A 0.000,B 0.000,C 90.000,E1 88.625} C_DIS
LIN {X -0.176,Y -566.560,Z 1171.283,A 0.000,B 0.000,C 90.000,E1 87.020} C_DIS
LIN {X 0.002,Y -567.588,Z 1171.274,A 0.000,B 0.000,C 90.000,E1 85.355} C_DIS
LIN {X 0.254,Y -568.706,Z 1171.265,A 0.000,B 0.000,C 90.000,E1 83.685} C_DIS
LIN {X 0.038,Y -569.773,Z 1171.256,A 0.000,B 0.000,C 90.000,E1 82.064} C_DIS
LIN {X 0.222,Y -570.541,Z 1171.248,A 0.000,B 0.000,C 90.000,E1 80.679} C_DIS
LIN {X 0.129,Y -571.399,Z 1171.239,A 0.000,B 0.000,C 90.000,E1 79.050} C_DIS
LIN {X 0.167,Y -572.242,Z 1171.230,A 0.000,B 0.000,C 90.000,E1 77.409} C_DIS
LIN {X -0.007,Y -573.211,Z 1171.220,A 0.000,B 0.000,C 90.000,E1 75.519} C_DIS
LIN {X 0.003,Y -573.825,Z 1171.212,A 0.000,B 0.000,C 90.000,E1 74.157} C_DIS
LIN {X 0.183,Y -574.971,Z 1171.201,A 0.000,B 0.000,C 90.000,E1 72.236} C_DIS
LIN {X -0.153,Y -576.621,Z 1171.188,A 0.000,B 0.000,C 90.000,E1 69.826} C_DIS
LIN {X 0.153,Y -578.669,Z 1171.174,A 0.000,B 0.000,C 90.000,E1 67.358} C_DIS
LIN {X -0.275,Y -580.021,Z 1171.167,A 0.000,B 0.000,C 90.000,E1 66.049} C_DIS
LIN {X -0.052,Y -581.539,Z 1171.158,A 0.000,B 0.000,C 90.000,E1 64.409} C_DIS
LIN {X -0.190,Y -583.304,Z 1171.147,A 0.000,B 0.000,C 90.000,E1 62.538} C_DIS
LIN {X -0.161,Y -584.790,Z 1171.138,A 0.000,B 0.000,C 90.000,E1 60.923} C_DIS
LIN {X 0.173,Y -586.209,Z 1171.130,A 0.000,B 0.000,C 90.000,E1 59.282} C_DIS
LIN {X 0.145,Y -587.235,Z 1171.122,A 0.000,B 0.000,C 90.000,E1 57.946} C_DIS
LIN {X -0.237,Y -588.012,Z 1171.116,A 0.000,B 0.000,C 90.000,E1 56.914} C_DIS
LIN {X 0.214,Y -588.738,Z 1171.110,A 0.000,B 0.000,C 90.000,E1 55.801} C_DIS
LIN {X 0.058,Y -589.616,Z 1171.103,A 0.000,B 0.000,C 90.000,E1 54.482} C_DIS
LIN {X -0.155,Y -590.774,Z 1171.092,A 0.000,B 0.000,C 90.000,E1 52.637} C_DIS
LIN {X 0.380,Y -591.868,Z 1171.082,A 0.000,B 0.000,C 90.000,E1 50.723} C_DIS
LIN {X -0.280,Y -592.276,Z 1171.078,A 0.000,B 0.000,C 90.000,E1 49.989} C_DIS
LIN {X 0.015,Y -592.772,Z 1171.069,A 0.000,B 0.000,C 90.000,E1 48.366} C_DIS
LIN {X -0.278,Y -593.025,Z 1171.061,A 0.000,B 0.000,C 90.000,E1 47.067} C_DIS
LIN {X 0.294,Y -593.104,Z 1171.057,A 0.000,B 0.000,C 90.000,E1 46.215} C_DIS
LIN {X 0.207,Y -592.958,Z 1171.051,A 0.000,B 0.000,C 90.000,E1 45.162} C_DIS
LIN {X -0.114,Y -592.591,Z 1171.044,A 0.000,B 0.000,C 90.000,E1 43.866} C_DIS
LIN {X 0.217,Y -592.013,Z 1171.038,A 0.000,B 0.000,C 90.000,E1 42.771} C_DIS
LIN {X -0.094,Y -591.144,Z 1171.030,A 0.000,B 0.000,C 90.000,E1 41.472} C_DIS
LIN {X 0.009,Y -590.521,Z 1171.026,A 0.000,B 0.000,C 90.000,E1 40.663} C_DIS
LIN {X -0.264,Y -589.127,Z 1171.019,A 0.000,B 0.000,C 90.000,E1 39.358} C_DIS
LIN {X -0.118,Y -588.158,Z 1171.014,A 0.000,B 0.000,C 90.000,E1 38.543} C_DIS
LIN {X -0.063,Y -586.291,Z 1171.007,A 0.000,B 0.000,C 90.000,E1 37.202} C_DIS
LIN {X -0.126,Y -584.437,Z 1171.001,A 0.000,B 0.000,C 90.000,E1 36.137} C_DIS
LIN {X -0.098,Y -583.338,Z 1170.998,A 0.000,B 0.000,C 90.000,E1 35.598} C_DIS
LIN {X -0.198,Y -580.985,Z 1170.992,A 0.000,B 0.000,C 90.000,E1 34.532} C_DIS
LIN {X -0.021,Y -578.712,Z 1170.987,A 0.000,B 0.000,C 90.000,E1 33.706} C_DIS
LIN {X -0.030,Y -575.374,Z 1170.981,A 0.000,B 0.000,C 90.000,E1 32.625} C_DIS
LIN {X -0.050,Y -573.451,Z 1170.978,A 0.000,B 0.000,C 90.000,E1 32.084} C_DIS
LIN {X -0.131,Y -568.903,Z 1170.972,A 0.000,B 0.000,C 90.000,E1 31.003} C_DIS
LIN {X -0.096,Y -565.171,Z 1170.968,A 0.000,B 0.000,C 90.000,E1 30.178} C_DIS
LIN {X 0.192,Y -561.621,Z 1170.964,A 0.000,B 0.000,C 90.000,E1 29.461} C_DIS
LIN {X -0.208,Y -558.613,Z 1170.961,A 0.000,B 0.000,C 90.000,E1 28.949} C_DIS
LIN {X -0.191,Y -552.932,Z 1170.955,A 0.000,B 0.000,C 90.000,E1 27.975} C_DIS
LIN {X -0.012,Y -548.479,Z 1170.951,A 0.000,B 0.000,C 90.000,E1 27.257} C_DIS
LIN {X -0.001,Y -544.660,Z 1170.948,A 0.000,B 0.000,C 90.000,E1 26.693} C_DIS
LIN {X 0.227,Y -540.574,Z 1170.945,A 0.000,B 0.000,C 90.000,E1 26.104} C_DIS
LIN {X 0.185,Y -536.183,Z 1170.942,A 0.000,B 0.000,C 90.000,E1 25.540} C_DIS
LIN {X 0.115,Y -531.528,Z 1170.939,A 0.000,B 0.000,C 90.000,E1 24.975} C_DIS
LIN {X 0.082,Y -525.476,Z 1170.935,A 0.000,B 0.000,C 90.000,E1 24.259} C_DIS
LIN {X -0.082,Y -519.119,Z 1170.931,A 0.000,B 0.000,C 90.000,E1 23.567} C_DIS
LIN {X -0.151,Y -512.825,Z 1170.927,A 0.000,B 0.000,C 90.000,E1 22.898} C_DIS
LIN {X -0.011,Y -508.763,Z 1170.925,A 0.000,B 0.000,C 90.000,E1 22.461} C_DIS
LIN {X -0.112,Y -500.599,Z 1170.920,A 0.000,B 0.000,C 90.000,E1 21.663} C_DIS
LIN {X -0.128,Y -490.734,Z 1170.915,A 0.000,B 0.000,C 90.000,E1 20.737} C_DIS
LIN {X -0.137,Y -481.991,Z 1170.911,A 0.000,B 0.000,C 90.000,E1 19.939} C_DIS
LIN {X 0.104,Y -470.193,Z 1170.905,A 0.000,B 0.000,C 90.000,E1 18.852} C_DIS
LIN {X -0.184,Y -458.222,Z 1170.899,A 0.000,B 0.000,C 90.000,E1 17.819} C_DIS
LIN {X 0.128,Y -448.094,Z 1170.894,A 0.000,B 0.000,C 90.000,E1 16.858} C_DIS
LIN {X -0.047,Y -428.147,Z 1170.883,A 0.000,B 0.000,C 90.000,E1 14.898} C_DIS
LIN {X -0.165,Y -415.680,Z 1170.875,A 0.000,B 0.000,C 90.000,E1 13.536} C_DIS
LIN {X 0.173,Y -407.811,Z 1170.870,A 0.000,B 0.000,C 90.000,E1 12.535} C_DIS
LIN {X 0.016,Y -400.143,Z 1170.864,A 0.000,B 0.000,C 90.000,E1 11.535} C_DIS
LIN {X -0.114,Y -395.835,Z 1170.860,A 0.000,B 0.000,C 90.000,E1 10.894} C_DIS
LIN {X 0.220,Y -393.552,Z 1170.858,A 0.000,B 0.000,C 90.000,E1 10.366} C_DIS
LIN {X 0.107,Y -392.710,Z 1170.856,A 0.000,B 0.000,C 90.000,E1 10.018} C_DIS
LIN {X 0.069,Y -392.709,Z 1170.856,A 0.000,B 0.000,C 90.000,E1 10.018} C_DIS
LIN {X -0.080,Y -393.192,Z 1170.853,A 0.000,B 0.000,C 90.000,E1 9.613} C_DIS
LIN {X -0.162,Y -394.906,Z 1170.849,A 0.000,B 0.000,C 90.000,E1 8.916} C_DIS
LIN {X -0.205,Y -397.888,Z 1170.845,A 0.000,B 0.000,C 90.000,E1 8.049} C_DIS
LIN {X 0.026,Y -402.325,Z 1170.839,A 0.000,B 0.000,C 90.000,E1 7.004} C_DIS
LIN {X -0.077,Y -406.345,Z 1170.836,A 0.000,B 0.000,C 90.000,E1 6.429} C_DIS
LIN {X -0.101,Y -407.735,Z 1170.835,A 0.000,B 0.000,C 90.000,E1 6.258} C_DIS
LIN {X 0.186,Y -411.060,Z 1170.833,A 0.000,B 0.000,C 90.000,E1 5.910} C_DIS
LIN {X 0.051,Y -418.631,Z 1170.830,A 0.000,B 0.000,C 90.000,E1 5.334} C_DIS
LIN {X -0.021,Y -426.489,Z 1170.826,A 0.000,B 0.000,C 90.000,E1 4.759} C_DIS
LIN {X 0.056,Y -450.697,Z 1170.817,A 0.000,B 0.000,C 90.000,E1 2.980} C_DIS
LIN {X 0.130,Y -465.175,Z 1170.811,A 0.000,B 0.000,C 90.000,E1 1.949} C_DIS
LIN {X -0.233,Y -474.665,Z 1170.807,A 0.000,B 0.000,C 90.000,E1 1.318} C_DIS
LIN {X 0.236,Y -480.884,Z 1170.805,A 0.000,B 0.000,C 90.000,E1 0.802} C_DIS
LIN {X 0.122,Y -487.022,Z 1170.802,A 0.000,B 0.000,C 90.000,E1 0.344} C_DIS
LIN {X 0.000,Y -491.513,Z 1170.800,A 0.000,B 0.000,C 90.000,E1 360.000} C_DIS
LIN {X 0.021,Y -496.987,Z 1170.797,A 0.000,B 0.000,C 90.000,E1 359.542} C_DIS
LIN {X -0.059,Y -503.877,Z 1170.794,A 0.000,B 0.000,C 90.000,E1 358.912} C_DIS
LIN {X -0.210,Y -511.834,Z 1170.789,A 0.000,B 0.000,C 90.000,E1 358.108} C_DIS
LIN {X 0.009,Y -518.166,Z 1170.785,A 0.000,B 0.000,C 90.000,E1 357.364} C_DIS
LIN {X -0.089,Y -523.082,Z 1170.782,A 0.000,B 0.000,C 90.000,E1 356.788} C_DIS
LIN {X 0.062,Y -528.585,Z 1170.778,A 0.000,B 0.000,C 90.000,E1 356.045} C_DIS
LIN {X -0.237,Y -533.581,Z 1170.774,A 0.000,B 0.000,C 90.000,E1 355.355} C_DIS
LIN {X -0.220,Y -537.229,Z 1170.771,A 0.000,B 0.000,C 90.000,E1 354.780} C_DIS
LIN {X 0.094,Y -541.311,Z 1170.767,A 0.000,B 0.000,C 90.000,E1 354.033} C_DIS
LIN {X 0.168,Y -544.297,Z 1170.764,A 0.000,B 0.000,C 90.000,E1 353.457} C_DIS
LIN {X 0.068,Y -547.694,Z 1170.760,A 0.000,B 0.000,C 90.000,E1 352.761} C_DIS
LIN {X 0.188,Y -550.279,Z 1170.757,A 0.000,B 0.000,C 90.000,E1 352.186} C_DIS
LIN {X -0.114,Y -553.693,Z 1170.752,A 0.000,B 0.000,C 90.000,E1 351.376} C_DIS
LIN {X 0.254,Y -556.729,Z 1170.747,A 0.000,B 0.000,C 90.000,E1 350.500} C_DIS
LIN {X 0.017,Y -559.461,Z 1170.743,A 0.000,B 0.000,C 90.000,E1 349.690} C_DIS
LIN {X 0.059,Y -562.713,Z 1170.737,A 0.000,B 0.000,C 90.000,E1 348.578} C_DIS
LIN {X 0.152,Y -565.694,Z 1170.730,A 0.000,B 0.000,C 90.000,E1 347.465} C_DIS
LIN {X -0.271,Y -568.512,Z 1170.724,A 0.000,B 0.000,C 90.000,E1 346.408} C_DIS
LIN {X 0.217,Y -571.731,Z 1170.717,A 0.000,B 0.000,C 90.000,E1 344.991} C_DIS
LIN {X 0.014,Y -574.152,Z 1170.711,A 0.000,B 0.000,C 90.000,E1 343.921} C_DIS
LIN {X -0.152,Y -577.611,Z 1170.702,A 0.000,B 0.000,C 90.000,E1 342.308} C_DIS
LIN {X 0.275,Y -580.239,Z 1170.694,A 0.000,B 0.000,C 90.000,E1 340.913} C_DIS
LIN {X -0.191,Y -582.093,Z 1170.688,A 0.000,B 0.000,C 90.000,E1 339.880} C_DIS
LIN {X 0.116,Y -583.725,Z 1170.682,A 0.000,B 0.000,C 90.000,E1 338.773} C_DIS
LIN {X -0.094,Y -585.042,Z 1170.676,A 0.000,B 0.000,C 90.000,E1 337.720} C_DIS
LIN {X -0.161,Y -585.819,Z 1170.672,A 0.000,B 0.000,C 90.000,E1 336.922} C_DIS
LIN {X 0.007,Y -586.237,Z 1170.667,A 0.000,B 0.000,C 90.000,E1 336.102} C_DIS
LIN {X 0.303,Y -586.427,Z 1170.664,A 0.000,B 0.000,C 90.000,E1 335.537} C_DIS
LIN {X -0.298,Y -586.300,Z 1170.660,A 0.000,B 0.000,C 90.000,E1 334.793} C_DIS
LIN {X 0.131,Y -585.901,Z 1170.655,A 0.000,B 0.000,C 90.000,E1 333.948} C_DIS
LIN {X -0.104,Y -585.498,Z 1170.652,A 0.000,B 0.000,C 90.000,E1 333.435} C_DIS
LIN {X -0.065,Y -584.091,Z 1170.646,A 0.000,B 0.000,C 90.000,E1 332.359} C_DIS
LIN {X 0.215,Y -582.149,Z 1170.641,A 0.000,B 0.000,C 90.000,E1 331.257} C_DIS
LIN {X 0.096,Y -580.137,Z 1170.636,A 0.000,B 0.000,C 90.000,E1 330.461} C_DIS
LIN {X -0.040,Y -577.797,Z 1170.631,A 0.000,B 0.000,C 90.000,E1 329.665} C_DIS
LIN {X -0.188,Y -576.878,Z 1170.630,A 0.000,B 0.000,C 90.000,E1 329.410} C_DIS
LIN {X -0.280,Y -574.060,Z 1170.626,A 0.000,B 0.000,C 90.000,E1 328.742} C_DIS
LIN {X -0.097,Y -570.617,Z 1170.622,A 0.000,B 0.000,C 90.000,E1 328.043} C_DIS
LIN {X 0.136,Y -565.693,Z 1170.618,A 0.000,B 0.000,C 90.000,E1 327.199} C_DIS
LIN {X 0.143,Y -563.126,Z 1170.616,A 0.000,B 0.000,C 90.000,E1 326.786} C_DIS
LIN {X 0.229,Y -558.216,Z 1170.612,A 0.000,B 0.000,C 90.000,E1 326.087} C_DIS
LIN {X 0.273,Y -552.810,Z 1170.608,A 0.000,B 0.000,C 90.000,E1 325.388} C_DIS
LIN {X 0.214,Y -549.407,Z 1170.606,A 0.000,B 0.000,C 90.000,E1 324.975} C_DIS
LIN {X 0.056,Y -542.041,Z 1170.601,A 0.000,B 0.000,C 90.000,E1 324.149} C_DIS
LIN {X -0.246,Y -527.462,Z 1170.592,A 0.000,B 0.000,C 90.000,E1 322.557} C_DIS
LIN {X -0.268,Y -525.061,Z 1170.590,A 0.000,B 0.000,C 90.000,E1 322.271} C_DIS
LIN {X -0.050,Y -521.437,Z 1170.588,A 0.000,B 0.000,C 90.000,E1 321.743} C_DIS
LIN {X 0.002,Y -519.715,Z 1170.586,A 0.000,B 0.000,C 90.000,E1 321.412} C_DIS
LIN {X 0.141,Y -519.087,Z 1170.585,A 0.000,B 0.000,C 90.000,E1 321.251} C_DIS
LIN {X 0.023,Y -517.582,Z 1170.582,A 0.000,B 0.000,C 90.000,E1 320.803} C_DIS
LIN {X -0.037,Y -517.070,Z 1170.581,A 0.000,B 0.000,C 90.000,E1 320.517} C_DIS
LIN {X 0.280,Y -516.467,Z 1170.578,A 0.000,B 0.000,C 90.000,E1 319.908} C_DIS
LIN {X -0.253,Y -516.471,Z 1170.574,A 0.000,B 0.000,C 90.000,E1 319.380} C_DIS
LIN {X -0.119,Y -517.483,Z 1170.563,A 0.000,B 0.000,C 90.000,E1 317.310} C_DIS
LIN {X 0.183,Y -518.298,Z 1170.555,A 0.000,B 0.000,C 90.000,E1 315.810} C_DIS
LIN {X 0.131,Y -519.070,Z 1170.547,A 0.000,B 0.000,C 90.000,E1 314.352} C_DIS
LIN {X 0.084,Y -519.883,Z 1170.538,A 0.000,B 0.000,C 90.000,E1 312.894} C_DIS
LIN {X 0.015,Y -520.959,Z 1170.529,A 0.000,B 0.000,C 90.000,E1 311.148} C_DIS
LIN {X 0.023,Y -521.849,Z 1170.521,A 0.000,B 0.000,C 90.000,E1 309.688} C_DIS
LIN {X 0.021,Y -523.097,Z 1170.509,A 0.000,B 0.000,C 90.000,E1 307.649} C_DIS
LIN {X -0.188,Y -523.934,Z 1170.501,A 0.000,B 0.000,C 90.000,E1 306.217} C_DIS
LIN {X 0.065,Y -525.240,Z 1170.488,A 0.000,B 0.000,C 90.000,E1 303.865} C_DIS
LIN {X 0.028,Y -526.151,Z 1170.480,A 0.000,B 0.000,C 90.000,E1 302.418} C_DIS
LIN {X 0.086,Y -527.266,Z 1170.469,A 0.000,B 0.000,C 90.000,E1 300.384} C_DIS
LIN {X 0.186,Y -527.562,Z 1170.466,A 0.000,B 0.000,C 90.000,E1 299.795} C_DIS
LIN {X -0.214,Y -528.120,Z 1170.456,A 0.000,B 0.000,C 90.000,E1 298.103} C_DIS
LIN {X 0.168,Y -528.427,Z 1170.448,A 0.000,B 0.000,C 90.000,E1 296.616} C_DIS
LIN {X -0.158,Y -528.612,Z 1170.440,A 0.000,B 0.000,C 90.000,E1 295.207} C_DIS
LIN {X -0.226,Y -528.616,Z 1170.432,A 0.000,B 0.000,C 90.000,E1 293.770} C_DIS
LIN {X -0.110,Y -528.506,Z 1170.422,A 0.000,B 0.000,C 90.000,E1 292.025} C_DIS
LIN {X -0.202,Y -528.226,Z 1170.413,A 0.000,B 0.000,C 90.000,E1 290.301} C_DIS
LIN {X 0.187,Y -527.747,Z 1170.401,A 0.000,B 0.000,C 90.000,E1 288.236} C_DIS
LIN {X 0.225,Y -527.125,Z 1170.392,A 0.000,B 0.000,C 90.000,E1 286.496} C_DIS
LIN {X -0.072,Y -526.635,Z 1170.385,A 0.000,B 0.000,C 90.000,E1 285.371} C_DIS
LIN {X 0.139,Y -525.992,Z 1170.379,A 0.000,B 0.000,C 90.000,E1 284.189} C_DIS
LIN {X -0.135,Y -524.915,Z 1170.369,A 0.000,B 0.000,C 90.000,E1 282.479} C_DIS
LIN {X 0.052,Y -523.989,Z 1170.361,A 0.000,B 0.000,C 90.000,E1 281.007} C_DIS
LIN {X 0.029,Y -522.815,Z 1170.352,A 0.000,B 0.000,C 90.000,E1 279.265} C_DIS
LIN {X -0.025,Y -522.105,Z 1170.345,A 0.000,B 0.000,C 90.000,E1 278.106} C_DIS
LIN {X -0.164,Y -521.037,Z 1170.335,A 0.000,B 0.000,C 90.000,E1 276.372} C_DIS
LIN {X 0.131,Y -520.052,Z 1170.326,A 0.000,B 0.000,C 90.000,E1 274.588} C_DIS
LIN {X -0.215,Y -519.073,Z 1170.314,A 0.000,B 0.000,C 90.000,E1 272.579} C_DIS
LIN {X -0.087,Y -518.125,Z 1170.303,A 0.000,B 0.000,C 90.000,E1 270.516} C_DIS
LIN {X 0.069,Y -517.351,Z 1170.293,A 0.000,B 0.000,C 90.000,E1 268.740} C_DIS
END
